KUKA KRL program: EPS_2_25748_MH07A_A_20260121065905.src

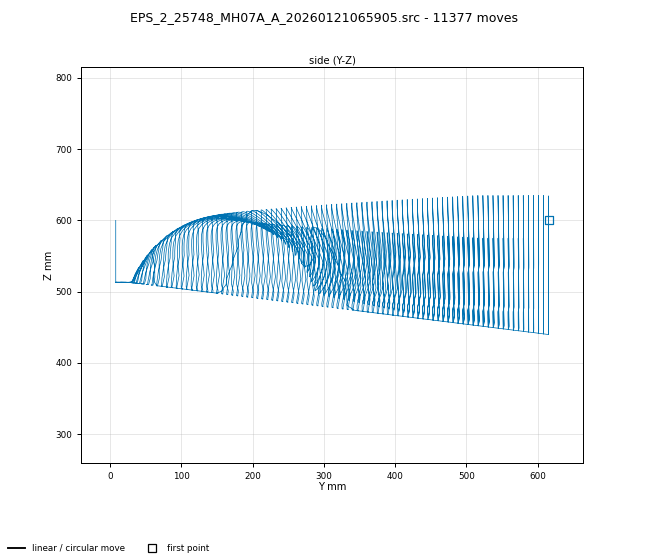
[picture p0: tool path of EPS_2_25748_MH07A_A_20260121065905.src, 11377 of 11379 moves have a stored position in this frame; points joined in program order, loops and branches not executed]
&ACCESS RVP
&REL 4
&COMMENT QRS 19112012
&PARAM EDITMASK = *
DEF PART()
EXT BAS (BAS_COMMAND :IN,REAL :IN )
INT I
BAS (#INITMOV,0 )

;KUKA QRS Post kuka4.cps  Date:22-06-2017 !

File_ID=3007

QRS_PRE_INIT()

;Init var - Until changes are made in qrs_pre_init
Outlet_Square_prg=0
Inlet_1_Square_prg=0
Inlet_2_Square_prg=0
Inlet_3_Square_prg=0
Inlet_4_Square_prg=0
Inlet_5_Square_prg=0

Outlet_1={X 0.000, Y 515.340, Z 534.500, B 0.000, E1 0.000 }
Inlet_1={X 0.000, Y 519.690, Z 474.500, B 0.000, E1 270.000 }
Outlet_1_type=201
Inlet_1_type=201
;QRS#1=Sidecore dimensions
;QRS#2=200-8" PVC SDR 35
;QRS#3=200-8" PVC SDR 35
;QRS#4=
;QRS#5=
;QRS#6=
;QRS#7=
;QRS#8=
;QRS#9=12-08 PSX
;QRS#10=12-08 PSX
;QRS#11=
;QRS#12=
;QRS#13=
;QRS#14=
;QRS#15=
;QRS#16=1220x127x914 3'
;QRS#17=EPS Height
;QRS#18=635
;QRS#19=*
;QRS#20= UPDATED VERSION 22-06-2017
;QRS#21=*
Outlet_Square=0100
Inlet_1_Square=0100
Inlet_2_Square=0
Inlet_3_Square=0
Inlet_4_Square=0
Inlet_5_Square=0
Mill_Square=1
Outlet_Square_Prg=204
Inlet_1_Square_prg=204

QRS_INIT()

$ADVANCE=5

; T1
PTP {E1 173.607,E2 173.607}
PTP {X 0,Y 615.507,A -85,B 0,C 180,E1 173.607,E2 173.607,E3 0,E4 0,E5 0,E6 0}
QRS_SPEED_INIT()
LIN {X 0,Y 615.507,Z 600,A -85,B 0,C 180,E1 173.607,E2 173.607,E3 0,E4 0,E5 0,E6 0} C_VEL
LIN {X 0,Y 615.507,Z 449.87,A -85,B 0,C 180,E1 173.607,E2 173.607} C_VEL
LIN {X 0,Y 615.507,Z 441.69,A -85,B 0,C 180,E1 173.607,E2 173.607} C_VEL
LIN {X 0,Y 615.491,Z 439.69,A -85,B 0,C 180,E1 173.421,E2 173.421} C_VEL
LIN {X 0,Y 615.486,Z 439.701,A -85,B 0,C 180,E1 170.801,E2 170.801} C_VEL
LIN {X 0,Y 615.477,Z 439.696,A -85,B 0,C 180,E1 168.139,E2 168.139} C_VEL
LIN {X 0,Y 615.49,Z 439.69,A -85,B 0,C 180,E1 165.451,E2 165.451} C_VEL
LIN {X 0,Y 615.491,Z 439.693,A -85,B 0,C 180,E1 162.729,E2 162.729} C_VEL
LIN {X 0,Y 615.49,Z 439.702,A -85,B 0,C 180,E1 159.967,E2 159.967} C_VEL
LIN {X 0,Y 615.486,Z 439.695,A -85,B 0,C 180,E1 157.155,E2 157.155} C_VEL
LIN {X 0,Y 615.48,Z 439.693,A -85,B 0,C 180,E1 154.284,E2 154.284} C_VEL
LIN {X 0,Y 615.491,Z 439.69,A -85,B 0,C 180,E1 151.549,E2 151.549} C_VEL
LIN {X 0,Y 615.491,Z 439.699,A -85,B 0,C 180,E1 148.914,E2 148.914} C_VEL
LIN {X 0,Y 615.485,Z 439.692,A -85,B 0,C 180,E1 146.466,E2 146.466} C_VEL
LIN {X 0,Y 615.489,Z 439.69,A -85,B 0,C 180,E1 143.575,E2 143.575} C_VEL
LIN {X 0,Y 615.484,Z 439.696,A -85,B 0,C 180,E1 140.938,E2 140.938} C_VEL
LIN {X 0,Y 615.486,Z 439.693,A -85,B 0,C 180,E1 138.526,E2 138.526} C_VEL
LIN {X 0,Y 615.493,Z 439.689,A -85,B 0,C 180,E1 135.85,E2 135.85} C_VEL
LIN {X 0,Y 615.481,Z 439.695,A -85,B 0,C 180,E1 133.046,E2 133.046} C_VEL
LIN {X 0,Y 615.493,Z 439.695,A -85,B 0,C 180,E1 130.089,E2 130.089} C_VEL
LIN {X 0,Y 615.492,Z 439.7,A -85,B 0,C 180,E1 127.242,E2 127.242} C_VEL
LIN {X 0,Y 615.491,Z 439.69,A -85,B 0,C 180,E1 124.7,E2 124.7} C_VEL
LIN {X 0,Y 615.491,Z 439.697,A -85,B 0,C 180,E1 122.331,E2 122.331} C_VEL
LIN {X 0,Y 615.499,Z 439.691,A -85,B 0,C 180,E1 119.796,E2 119.796} C_VEL
LIN {X 0,Y 615.486,Z 439.69,A -85,B 0,C 180,E1 117.044,E2 117.044} C_VEL
LIN {X 0,Y 615.483,Z 439.693,A -85,B 0,C 180,E1 114.272,E2 114.272} C_VEL
LIN {X 0,Y 615.48,Z 439.7,A -85,B 0,C 180,E1 111.432,E2 111.432} C_VEL
LIN {X 0,Y 615.488,Z 439.699,A -85,B 0,C 180,E1 108.603,E2 108.603} C_VEL
LIN {X 0,Y 615.489,Z 439.691,A -85,B 0,C 180,E1 105.905,E2 105.905} C_VEL
LIN {X 0,Y 615.482,Z 439.692,A -85,B 0,C 180,E1 103.201,E2 103.201} C_VEL
LIN {X 0,Y 615.488,Z 439.698,A -85,B 0,C 180,E1 100.527,E2 100.527} C_VEL
LIN {X 0,Y 615.494,Z 439.693,A -85,B 0,C 180,E1 97.875,E2 97.875} C_VEL
LIN {X 0,Y 615.482,Z 439.691,A -85,B 0,C 180,E1 95.241,E2 95.241} C_VEL
LIN {X 0,Y 615.484,Z 439.697,A -85,B 0,C 180,E1 92.618,E2 92.618} C_VEL
LIN {X 0,Y 615.491,Z 439.695,A -85,B 0,C 180,E1 90,E2 90} C_VEL
LIN {X 0,Y 615.478,Z 439.692,A -85,B 0,C 180,E1 87.382,E2 87.382} C_VEL
LIN {X 0,Y 615.482,Z 439.696,A -85,B 0,C 180,E1 84.759,E2 84.759} C_VEL
LIN {X 0,Y 615.488,Z 439.698,A -85,B 0,C 180,E1 82.124,E2 82.124} C_VEL
LIN {X 0,Y 615.478,Z 439.693,A -85,B 0,C 180,E1 79.473,E2 79.473} C_VEL
LIN {X 0,Y 615.48,Z 439.694,A -85,B 0,C 180,E1 76.798,E2 76.798} C_VEL
LIN {X 0,Y 615.486,Z 439.701,A -85,B 0,C 180,E1 74.095,E2 74.095} C_VEL
LIN {X 0,Y 615.483,Z 439.696,A -85,B 0,C 180,E1 71.354,E2 71.354} C_VEL
LIN {X 0,Y 615.477,Z 439.693,A -85,B 0,C 180,E1 68.568,E2 68.568} C_VEL
LIN {X 0,Y 615.478,Z 439.693,A -85,B 0,C 180,E1 65.727,E2 65.727} C_VEL
LIN {X 0,Y 615.486,Z 439.696,A -85,B 0,C 180,E1 62.956,E2 62.956} C_VEL
LIN {X 0,Y 615.497,Z 439.698,A -85,B 0,C 180,E1 60.205,E2 60.205} C_VEL
LIN {X 0,Y 615.479,Z 439.693,A -85,B 0,C 180,E1 57.542,E2 57.542} C_VEL
LIN {X 0,Y 615.499,Z 439.693,A -85,B 0,C 180,E1 55.185,E2 55.185} C_VEL
LIN {X 0,Y 615.48,Z 439.694,A -85,B 0,C 180,E1 52.757,E2 52.757} C_VEL
LIN {X 0,Y 615.476,Z 439.693,A -85,B 0,C 180,E1 49.913,E2 49.913} C_VEL
LIN {X 0,Y 615.499,Z 439.7,A -85,B 0,C 180,E1 47.648,E2 47.648} C_VEL
LIN {X 0,Y 615.484,Z 439.694,A -85,B 0,C 180,E1 44.931,E2 44.931} C_VEL
LIN {X 0,Y 615.488,Z 439.69,A -85,B 0,C 180,E1 42.08,E2 42.08} C_VEL
LIN {X 0,Y 615.481,Z 439.702,A -85,B 0,C 180,E1 39.751,E2 39.751} C_VEL
LIN {X 0,Y 615.487,Z 439.697,A -85,B 0,C 180,E1 36.936,E2 36.936} C_VEL
LIN {X 0,Y 615.48,Z 439.694,A -85,B 0,C 180,E1 35.617,E2 35.617} C_VEL
LIN {X 0,Y 615.483,Z 440.393,A -85,B 0,C 180,E1 34.7,E2 34.7} C_VEL
LIN {X 0,Y 615.494,Z 443.234,A -85,B 0,C 180,E1 32.331,E2 32.331} C_VEL
LIN {X 0,Y 615.487,Z 446.882,A -85,B 0,C 180,E1 29.407,E2 29.407} C_VEL
LIN {X 0,Y 615.481,Z 449.92,A -85,B 0,C 180,E1 27.043,E2 27.043} C_VEL
LIN {X 0,Y 615.493,Z 453.568,A -85,B 0,C 180,E1 24.272,E2 24.272} C_VEL
LIN {X 0,Y 615.494,Z 457.377,A -85,B 0,C 180,E1 21.432,E2 21.432} C_VEL
LIN {X 0,Y 615.494,Z 461.252,A -85,B 0,C 180,E1 18.605,E2 18.605} C_VEL
LIN {X 0,Y 615.476,Z 465.011,A -85,B 0,C 180,E1 15.906,E2 15.906} C_VEL
LIN {X 0,Y 615.493,Z 468.827,A -85,B 0,C 180,E1 13.201,E2 13.201} C_VEL
LIN {X 0,Y 615.484,Z 471.187,A -85,B 0,C 180,E1 11.548,E2 11.548} C_VEL
LIN {X 0,Y 615.485,Z 486.249,A -85,B 0,C 180,E1 11.193,E2 11.193} C_VEL
LIN {X 0,Y 615.481,Z 498.967,A -85,B 0,C 180,E1 10.749,E2 10.749} C_VEL
LIN {X 0,Y 615.483,Z 510.755,A -85,B 0,C 180,E1 10.195,E2 10.195} C_VEL
LIN {X 0,Y 615.498,Z 521.845,A -85,B 0,C 180,E1 9.53,E2 9.53} C_VEL
LIN {X 0,Y 615.498,Z 530.82,A -85,B 0,C 180,E1 8.868,E2 8.868} C_VEL
LIN {X 0,Y 615.498,Z 540.032,A -85,B 0,C 180,E1 8.041,E2 8.041} C_VEL
LIN {X 0,Y 615.499,Z 548.89,A -85,B 0,C 180,E1 7.058,E2 7.058} C_VEL
LIN {X 0,Y 615.497,Z 556.122,A -85,B 0,C 180,E1 6.063,E2 6.063} C_VEL
LIN {X 0,Y 615.497,Z 560.957,A -85,B 0,C 180,E1 5.241,E2 5.241} C_VEL
LIN {X 0,Y 615.493,Z 565.657,A -85,B 0,C 180,E1 4.257,E2 4.257} C_VEL
LIN {X 0,Y 615.495,Z 569.254,A -85,B 0,C 180,E1 3.273,E2 3.273} C_VEL
LIN {X 0,Y 615.496,Z 571.114,A -85,B 0,C 180,E1 2.618,E2 2.618} C_VEL
LIN {X 0,Y 615.497,Z 572.533,A -85,B 0,C 180,E1 1.963,E2 1.963} C_VEL
LIN {X 0,Y 615.497,Z 574.141,A -85,B 0,C 180,E1 0.654,E2 0.654} C_VEL
LIN {X 0,Y 615.494,Z 574.384,A -85,B 0,C 180,E1 0,E2 0} C_VEL
LIN {X 0,Y 615.495,Z 574.206,A -85,B 0,C 180,E1 -0.654,E2 -0.654} C_VEL
LIN {X 0,Y 615.496,Z 572.683,A -85,B 0,C 180,E1 -1.963,E2 -1.963} C_VEL
LIN {X 0,Y 615.498,Z 571.341,A -85,B 0,C 180,E1 -2.618,E2 -2.618} C_VEL
LIN {X 0,Y 615.498,Z 568.494,A -85,B 0,C 180,E1 -3.601,E2 -3.601} C_VEL
LIN {X 0,Y 615.498,Z 564.635,A -85,B 0,C 180,E1 -4.584,E2 -4.584} C_VEL
LIN {X 0,Y 615.499,Z 559.652,A -85,B 0,C 180,E1 -5.57,E2 -5.57} C_VEL
LIN {X 0,Y 615.496,Z 553.208,A -85,B 0,C 180,E1 -6.582,E2 -6.582} C_VEL
LIN {X 0,Y 615.497,Z 545.537,A -85,B 0,C 180,E1 -7.545,E2 -7.545} C_VEL
LIN {X 0,Y 615.498,Z 535.759,A -85,B 0,C 180,E1 -8.536,E2 -8.536} C_VEL
LIN {X 0,Y 615.498,Z 525.494,A -85,B 0,C 180,E1 -9.364,E2 -9.364} C_VEL
LIN {X 0,Y 615.479,Z 513.933,A -85,B 0,C 180,E1 -10.111,E2 -10.111} C_VEL
LIN {X 0,Y 615.482,Z 502.146,A -85,B 0,C 180,E1 -10.704,E2 -10.704} C_VEL
LIN {X 0,Y 615.483,Z 489.162,A -85,B 0,C 180,E1 -11.193,E2 -11.193} C_VEL
LIN {X 0,Y 615.487,Z 476.561,A -85,B 0,C 180,E1 -11.527,E2 -11.527} C_VEL
LIN {X 0,Y 615.484,Z 471.197,A -85,B 0,C 180,E1 -11.631,E2 -11.631} C_VEL
LIN {X 0,Y 615.476,Z 467.929,A -85,B 0,C 180,E1 -13.927,E2 -13.927} C_VEL
LIN {X 0,Y 615.487,Z 464.181,A -85,B 0,C 180,E1 -16.587,E2 -16.587} C_VEL
LIN {X 0,Y 615.489,Z 460.369,A -85,B 0,C 180,E1 -19.338,E2 -19.338} C_VEL
LIN {X 0,Y 615.479,Z 456.548,A -85,B 0,C 180,E1 -22.137,E2 -22.137} C_VEL
LIN {X 0,Y 615.491,Z 453.686,A -85,B 0,C 180,E1 -24.272,E2 -24.272} C_VEL
LIN {X 0,Y 615.481,Z 449.862,A -85,B 0,C 180,E1 -27.178,E2 -27.178} C_VEL
LIN {X 0,Y 615.497,Z 446.505,A -85,B 0,C 180,E1 -29.796,E2 -29.796} C_VEL
LIN {X 0,Y 615.489,Z 443.245,A -85,B 0,C 180,E1 -32.457,E2 -32.457} C_VEL
LIN {X 0,Y 615.488,Z 440.551,A -85,B 0,C 180,E1 -34.815,E2 -34.815} C_VEL
LIN {X 0,Y 615.478,Z 439.698,A -85,B 0,C 180,E1 -35.832,E2 -35.832} C_VEL
LIN {X 0,Y 615.491,Z 439.697,A -85,B 0,C 180,E1 -38.068,E2 -38.068} C_VEL
LIN {X 0,Y 615.479,Z 439.698,A -85,B 0,C 180,E1 -40.607,E2 -40.607} C_VEL
LIN {X 0,Y 615.498,Z 439.693,A -85,B 0,C 180,E1 -43.244,E2 -43.244} C_VEL
LIN {X 0,Y 615.483,Z 439.698,A -85,B 0,C 180,E1 -46.003,E2 -46.003} C_VEL
LIN {X 0,Y 615.493,Z 439.697,A -85,B 0,C 180,E1 -48.905,E2 -48.905} C_VEL
LIN {X 0,Y 615.492,Z 439.701,A -85,B 0,C 180,E1 -51.096,E2 -51.096} C_VEL
LIN {X 0,Y 615.484,Z 439.703,A -85,B 0,C 180,E1 -53.575,E2 -53.575} C_VEL
LIN {X 0,Y 615.486,Z 439.895,A -85,B 0,C 180,E1 -54.484,E2 -54.484} C_VEL
LIN {X 0,Y 615.486,Z 448.578,A -85,B 0,C 180,E1 -57.154,E2 -57.154} C_VEL
LIN {X 0,Y 615.48,Z 457.828,A -85,B 0,C 180,E1 -59.839,E2 -59.839} C_VEL
LIN {X 0,Y 615.481,Z 467.078,A -85,B 0,C 180,E1 -62.454,E2 -62.454} C_VEL
LIN {X 0,Y 615.488,Z 476.316,A -85,B 0,C 180,E1 -65.008,E2 -65.008} C_VEL
LIN {X 0,Y 615.482,Z 486.871,A -85,B 0,C 180,E1 -67.863,E2 -67.863} C_VEL
LIN {X 0,Y 615.475,Z 497.419,A -85,B 0,C 180,E1 -70.662,E2 -70.662} C_VEL
LIN {X 0,Y 615.48,Z 507.958,A -85,B 0,C 180,E1 -73.413,E2 -73.413} C_VEL
LIN {X 0,Y 615.493,Z 518.494,A -85,B 0,C 180,E1 -76.126,E2 -76.126} C_VEL
LIN {X 0,Y 615.487,Z 527.208,A -85,B 0,C 180,E1 -78.348,E2 -78.348} C_VEL
LIN {X 0,Y 615.496,Z 541.817,A -85,B 0,C 180,E1 -78.64,E2 -78.64} C_VEL
LIN {X 0,Y 615.49,Z 554.557,A -85,B 0,C 180,E1 -79.036,E2 -79.036} C_VEL
LIN {X 0,Y 615.477,Z 566.765,A -85,B 0,C 180,E1 -79.556,E2 -79.556} C_VEL
LIN {X 0,Y 615.491,Z 577.386,A -85,B 0,C 180,E1 -80.138,E2 -80.138} C_VEL
LIN {X 0,Y 615.498,Z 588.23,A -85,B 0,C 180,E1 -80.884,E2 -80.884} C_VEL
LIN {X 0,Y 615.497,Z 598.81,A -85,B 0,C 180,E1 -81.794,E2 -81.794} C_VEL
LIN {X 0,Y 615.498,Z 606.605,A -85,B 0,C 180,E1 -82.619,E2 -82.619} C_VEL
LIN {X 0,Y 615.496,Z 614.202,A -85,B 0,C 180,E1 -83.608,E2 -83.608} C_VEL
LIN {X 0,Y 615.498,Z 621.204,A -85,B 0,C 180,E1 -84.759,E2 -84.759} C_VEL
LIN {X 0,Y 615.493,Z 625.851,A -85,B 0,C 180,E1 -85.743,E2 -85.743} C_VEL
LIN {X 0,Y 615.495,Z 629.398,A -85,B 0,C 180,E1 -86.727,E2 -86.727} C_VEL
LIN {X 0,Y 615.497,Z 631.233,A -85,B 0,C 180,E1 -87.382,E2 -87.382} C_VEL
LIN {X 0,Y 615.497,Z 632.608,A -85,B 0,C 180,E1 -88.037,E2 -88.037} C_VEL
LIN {X 0,Y 615.496,Z 634.173,A -85,B 0,C 180,E1 -89.346,E2 -89.346} C_VEL
LIN {X 0,Y 615.494,Z 634.389,A -85,B 0,C 180,E1 -90,E2 -90} C_VEL
LIN {X 0,Y 615.496,Z 633.58,A -85,B 0,C 180,E1 -91.309,E2 -91.309} C_VEL
LIN {X 0,Y 615.497,Z 632.608,A -85,B 0,C 180,E1 -91.963,E2 -91.963} C_VEL
LIN {X 0,Y 615.497,Z 631.233,A -85,B 0,C 180,E1 -92.618,E2 -92.618} C_VEL
LIN {X 0,Y 615.496,Z 628.35,A -85,B 0,C 180,E1 -93.601,E2 -93.601} C_VEL
LIN {X 0,Y 615.498,Z 624.442,A -85,B 0,C 180,E1 -94.584,E2 -94.584} C_VEL
LIN {X 0,Y 615.499,Z 619.405,A -85,B 0,C 180,E1 -95.57,E2 -95.57} C_VEL
LIN {X 0,Y 615.497,Z 612.869,A -85,B 0,C 180,E1 -96.583,E2 -96.583} C_VEL
LIN {X 0,Y 615.497,Z 605.133,A -85,B 0,C 180,E1 -97.545,E2 -97.545} C_VEL
LIN {X 0,Y 615.498,Z 597.045,A -85,B 0,C 180,E1 -98.371,E2 -98.371} C_VEL
LIN {X 0,Y 615.499,Z 587.168,A -85,B 0,C 180,E1 -99.199,E2 -99.199} C_VEL
LIN {X 0,Y 615.488,Z 575.982,A -85,B 0,C 180,E1 -99.945,E2 -99.945} C_VEL
LIN {X 0,Y 615.478,Z 565.025,A -85,B 0,C 180,E1 -100.527,E2 -100.527} C_VEL
LIN {X 0,Y 615.494,Z 552.486,A -85,B 0,C 180,E1 -101.04,E2 -101.04} C_VEL
LIN {X 0,Y 615.495,Z 540.065,A -85,B 0,C 180,E1 -101.401,E2 -101.401} C_VEL
LIN {X 0,Y 615.487,Z 527.209,A -85,B 0,C 180,E1 -101.652,E2 -101.652} C_VEL
LIN {X 0,Y 615.48,Z 517.063,A -85,B 0,C 180,E1 -104.242,E2 -104.242} C_VEL
LIN {X 0,Y 615.495,Z 506.638,A -85,B 0,C 180,E1 -106.928,E2 -106.928} C_VEL
LIN {X 0,Y 615.485,Z 496.105,A -85,B 0,C 180,E1 -109.685,E2 -109.685} C_VEL
LIN {X 0,Y 615.477,Z 486.101,A -85,B 0,C 180,E1 -112.343,E2 -112.343} C_VEL
LIN {X 0,Y 615.489,Z 476.316,A -85,B 0,C 180,E1 -114.992,E2 -114.992} C_VEL
LIN {X 0,Y 615.481,Z 467.079,A -85,B 0,C 180,E1 -117.546,E2 -117.546} C_VEL
LIN {X 0,Y 615.483,Z 457.829,A -85,B 0,C 180,E1 -120.16,E2 -120.16} C_VEL
LIN {X 0,Y 615.489,Z 448.579,A -85,B 0,C 180,E1 -122.846,E2 -122.846} C_VEL
LIN {X 0,Y 615.486,Z 439.694,A -85,B 0,C 180,E1 -125.541,E2 -125.541} C_VEL
LIN {X 0,Y 615.485,Z 439.697,A -85,B 0,C 180,E1 -128.069,E2 -128.069} C_VEL
LIN {X 0,Y 615.484,Z 439.691,A -85,B 0,C 180,E1 -130.607,E2 -130.607} C_VEL
LIN {X 0,Y 615.477,Z 439.698,A -85,B 0,C 180,E1 -133.246,E2 -133.246} C_VEL
LIN {X 0,Y 615.49,Z 439.7,A -85,B 0,C 180,E1 -136.002,E2 -136.002} C_VEL
LIN {X 0,Y 615.485,Z 439.691,A -85,B 0,C 180,E1 -138.526,E2 -138.526} C_VEL
LIN {X 0,Y 615.478,Z 439.697,A -85,B 0,C 180,E1 -141.095,E2 -141.095} C_VEL
LIN {X 0,Y 615.488,Z 439.695,A -85,B 0,C 180,E1 -143.575,E2 -143.575} C_VEL
LIN {X 0,Y 615.484,Z 439.692,A -85,B 0,C 180,E1 -146.466,E2 -146.466} C_VEL
LIN {X 0,Y 615.478,Z 439.694,A -85,B 0,C 180,E1 -149.08,E2 -149.08} C_VEL
LIN {X 0,Y 615.491,Z 439.698,A -85,B 0,C 180,E1 -151.549,E2 -151.549} C_VEL
LIN {X 0,Y 615.485,Z 439.694,A -85,B 0,C 180,E1 -154.432,E2 -154.432} C_VEL
LIN {X 0,Y 615.475,Z 439.693,A -85,B 0,C 180,E1 -157.155,E2 -157.155} C_VEL
LIN {X 0,Y 615.491,Z 439.701,A -85,B 0,C 180,E1 -159.443,E2 -159.443} C_VEL
LIN {X 0,Y 615.477,Z 439.693,A -85,B 0,C 180,E1 -162.043,E2 -162.043} C_VEL
LIN {X 0,Y 615.486,Z 439.691,A -85,B 0,C 180,E1 -164.774,E2 -164.774} C_VEL
LIN {X 0,Y 615.489,Z 439.697,A -85,B 0,C 180,E1 -167.47,E2 -167.47} C_VEL
LIN {X 0,Y 615.479,Z 439.697,A -85,B 0,C 180,E1 -170.138,E2 -170.138} C_VEL
LIN {X 0,Y 615.483,Z 439.691,A -85,B 0,C 180,E1 -172.784,E2 -172.784} C_VEL
LIN {X 0,Y 615.491,Z 439.694,A -85,B 0,C 180,E1 -175.416,E2 -175.416} C_VEL
LIN {X 0,Y 615.482,Z 439.699,A -85,B 0,C 180,E1 -178.037,E2 -178.037} C_VEL
LIN {X 0,Y 615.488,Z 439.69,A -85,B 0,C 180,E1 -180.654,E2 -180.654} C_VEL
LIN {X 0,Y 615.485,Z 439.694,A -85,B 0,C 180,E1 -183.273,E2 -183.273} C_VEL
LIN {X 0,Y 615.485,Z 439.7,A -85,B 0,C 180,E1 -185.899,E2 -185.899} C_VEL
LIN {X 0,Y 615.491,Z 439.69,A -85,B 0,C 180,E1 -186.579,E2 -186.579} C_VEL
LIN {X 0,Y 614.811,Z 439.842,A -85,B 0,C 180,E1 -187.125,E2 -187.125} C_VEL
LIN {X 0,Y 611.975,Z 440.254,A -85,B 0,C 180,E1 -188.011,E2 -188.011} C_VEL
LIN {X 0,Y 609.584,Z 440.567,A -85,B 0,C 180,E1 -188.724,E2 -188.724} C_VEL
LIN {X 0,Y 608.548,Z 440.685,A -85,B 0,C 180,E1 -189.273,E2 -189.273} C_VEL
LIN {X 0,Y 608.457,Z 440.693,A -85,B 0,C 180,E1 -189.459,E2 -189.459} C_VEL
LIN {X 0,Y 608.457,Z 440.694,A -85,B 0,C 180,E1 -192,E2 -192} C_VEL
LIN {X 0,Y 608.478,Z 440.689,A -85,B 0,C 180,E1 -194.721,E2 -194.721} C_VEL
LIN {X 0,Y 608.453,Z 440.692,A -85,B 0,C 180,E1 -197.477,E2 -197.477} C_VEL
LIN {X 0,Y 608.465,Z 440.693,A -85,B 0,C 180,E1 -200.274,E2 -200.274} C_VEL
LIN {X 0,Y 608.462,Z 440.69,A -85,B 0,C 180,E1 -202.477,E2 -202.477} C_VEL
LIN {X 0,Y 608.448,Z 440.693,A -85,B 0,C 180,E1 -205.301,E2 -205.301} C_VEL
LIN {X 0,Y 608.449,Z 440.694,A -85,B 0,C 180,E1 -207.518,E2 -207.518} C_VEL
LIN {X 0,Y 608.464,Z 440.691,A -85,B 0,C 180,E1 -209.971,E2 -209.971} C_VEL
LIN {X 0,Y 608.463,Z 440.692,A -85,B 0,C 180,E1 -212.88,E2 -212.88} C_VEL
LIN {X 0,Y 608.446,Z 440.694,A -85,B 0,C 180,E1 -215.278,E2 -215.278} C_VEL
LIN {X 0,Y 608.469,Z 440.69,A -85,B 0,C 180,E1 -217.747,E2 -217.747} C_VEL
LIN {X 0,Y 608.448,Z 440.699,A -85,B 0,C 180,E1 -220.328,E2 -220.328} C_VEL
LIN {X 0,Y 608.452,Z 440.693,A -85,B 0,C 180,E1 -222.96,E2 -222.96} C_VEL
LIN {X 0,Y 608.45,Z 440.692,A -85,B 0,C 180,E1 -225.737,E2 -225.737} C_VEL
LIN {X 0,Y 608.457,Z 440.692,A -85,B 0,C 180,E1 -228.659,E2 -228.659} C_VEL
LIN {X 0,Y 608.466,Z 440.691,A -85,B 0,C 180,E1 -231.761,E2 -231.761} C_VEL
LIN {X 0,Y 608.451,Z 440.693,A -85,B 0,C 180,E1 -233.955,E2 -233.955} C_VEL
LIN {X 0,Y 608.453,Z 440.693,A -85,B 0,C 180,E1 -236.329,E2 -236.329} C_VEL
LIN {X 0,Y 608.451,Z 440.694,A -85,B 0,C 180,E1 -238.733,E2 -238.733} C_VEL
LIN {X 0,Y 608.47,Z 440.689,A -85,B 0,C 180,E1 -241.382,E2 -241.382} C_VEL
LIN {X 0,Y 608.446,Z 440.696,A -85,B 0,C 180,E1 -243.965,E2 -243.965} C_VEL
LIN {X 0,Y 608.467,Z 440.69,A -85,B 0,C 180,E1 -246.155,E2 -246.155} C_VEL
LIN {X 0,Y 608.457,Z 440.691,A -85,B 0,C 180,E1 -249.019,E2 -249.019} C_VEL
LIN {X 0,Y 608.457,Z 440.694,A -85,B 0,C 180,E1 -251.828,E2 -251.828} C_VEL
LIN {X 0,Y 608.473,Z 440.695,A -85,B 0,C 180,E1 -254.594,E2 -254.594} C_VEL
LIN {X 0,Y 608.472,Z 440.69,A -85,B 0,C 180,E1 -257.323,E2 -257.323} C_VEL
LIN {X 0,Y 608.462,Z 440.69,A -85,B 0,C 180,E1 -260.023,E2 -260.023} C_VEL
LIN {X 0,Y 608.466,Z 440.693,A -85,B 0,C 180,E1 -262.701,E2 -262.701} C_VEL
LIN {X 0,Y 608.452,Z 440.695,A -85,B 0,C 180,E1 -265.362,E2 -265.362} C_VEL
LIN {X 0,Y 608.468,Z 440.69,A -85,B 0,C 180,E1 -268.014,E2 -268.014} C_VEL
LIN {X 0,Y 608.475,Z 440.69,A -85,B 0,C 180,E1 -270.662,E2 -270.662} C_VEL
LIN {X 0,Y 608.48,Z 440.694,A -85,B 0,C 180,E1 -273.311,E2 -273.311} C_VEL
LIN {X 0,Y 608.467,Z 440.69,A -85,B 0,C 180,E1 -275.967,E2 -275.967} C_VEL
LIN {X 0,Y 608.452,Z 440.692,A -85,B 0,C 180,E1 -278.636,E2 -278.636} C_VEL
LIN {X 0,Y 608.486,Z 440.692,A -85,B 0,C 180,E1 -281.324,E2 -281.324} C_VEL
LIN {X 0,Y 608.476,Z 440.692,A -85,B 0,C 180,E1 -284.037,E2 -284.037} C_VEL
LIN {X 0,Y 608.444,Z 440.693,A -85,B 0,C 180,E1 -286.784,E2 -286.784} C_VEL
LIN {X 0,Y 608.45,Z 440.692,A -85,B 0,C 180,E1 -289.571,E2 -289.571} C_VEL
LIN {X 0,Y 608.465,Z 440.692,A -85,B 0,C 180,E1 -292.406,E2 -292.406} C_VEL
LIN {X 0,Y 608.453,Z 440.692,A -85,B 0,C 180,E1 -294.571,E2 -294.571} C_VEL
LIN {X 0,Y 608.477,Z 440.69,A -85,B 0,C 180,E1 -297.206,E2 -297.206} C_VEL
LIN {X 0,Y 608.472,Z 440.695,A -85,B 0,C 180,E1 -299.971,E2 -299.971} C_VEL
LIN {X 0,Y 608.455,Z 440.696,A -85,B 0,C 180,E1 -302.88,E2 -302.88} C_VEL
LIN {X 0,Y 608.447,Z 440.692,A -85,B 0,C 180,E1 -305.278,E2 -305.278} C_VEL
LIN {X 0,Y 608.467,Z 440.695,A -85,B 0,C 180,E1 -307.747,E2 -307.747} C_VEL
LIN {X 0,Y 608.444,Z 440.694,A -85,B 0,C 180,E1 -310.328,E2 -310.328} C_VEL
LIN {X 0,Y 608.45,Z 440.692,A -85,B 0,C 180,E1 -312.96,E2 -312.96} C_VEL
LIN {X 0,Y 608.46,Z 440.694,A -85,B 0,C 180,E1 -315.736,E2 -315.736} C_VEL
LIN {X 0,Y 608.465,Z 440.696,A -85,B 0,C 180,E1 -318.658,E2 -318.658} C_VEL
LIN {X 0,Y 608.466,Z 440.696,A -85,B 0,C 180,E1 -321.76,E2 -321.76} C_VEL
LIN {X 0,Y 608.449,Z 440.692,A -85,B 0,C 180,E1 -323.955,E2 -323.955} C_VEL
LIN {X 0,Y 608.423,Z 440.996,A -85,B 0,C 180,E1 -325.099,E2 -325.099} C_VEL
LIN {X 0,Y 608.435,Z 443.838,A -85,B 0,C 180,E1 -327.482,E2 -327.482} C_VEL
LIN {X 0,Y 608.444,Z 447.196,A -85,B 0,C 180,E1 -330.219,E2 -330.219} C_VEL
LIN {X 0,Y 608.427,Z 450.493,A -85,B 0,C 180,E1 -332.803,E2 -332.803} C_VEL
LIN {X 0,Y 608.423,Z 453.921,A -85,B 0,C 180,E1 -335.427,E2 -335.427} C_VEL
LIN {X 0,Y 608.418,Z 457.764,A -85,B 0,C 180,E1 -338.306,E2 -338.306} C_VEL
LIN {X 0,Y 608.424,Z 461.607,A -85,B 0,C 180,E1 -341.129,E2 -341.129} C_VEL
LIN {X 0,Y 608.421,Z 465.45,A -85,B 0,C 180,E1 -343.905,E2 -343.905} C_VEL
LIN {X 0,Y 608.432,Z 469.294,A -85,B 0,C 180,E1 -346.643,E2 -346.643} C_VEL
LIN {X 0,Y 608.429,Z 471.666,A -85,B 0,C 180,E1 -348.316,E2 -348.316} C_VEL
LIN {X 0,Y 608.53,Z 487.61,A -85,B 0,C 180,E1 -348.714,E2 -348.714} C_VEL
LIN {X 0,Y 608.503,Z 500.162,A -85,B 0,C 180,E1 -349.171,E2 -349.171} C_VEL
LIN {X 0,Y 608.48,Z 512.497,A -85,B 0,C 180,E1 -349.771,E2 -349.771} C_VEL
LIN {X 0,Y 608.488,Z 523.302,A -85,B 0,C 180,E1 -350.443,E2 -350.443} C_VEL
LIN {X 0,Y 608.477,Z 533.075,A -85,B 0,C 180,E1 -351.197,E2 -351.197} C_VEL
LIN {X 0,Y 608.46,Z 541.974,A -85,B 0,C 180,E1 -352.033,E2 -352.033} C_VEL
LIN {X 0,Y 608.465,Z 550.661,A -85,B 0,C 180,E1 -353.034,E2 -353.034} C_VEL
LIN {X 0,Y 608.439,Z 557.592,A -85,B 0,C 180,E1 -354.033,E2 -354.033} C_VEL
LIN {X 0,Y 608.436,Z 563.146,A -85,B 0,C 180,E1 -355.03,E2 -355.03} C_VEL
LIN {X 0,Y 608.434,Z 567.508,A -85,B 0,C 180,E1 -356.026,E2 -356.026} C_VEL
LIN {X 0,Y 608.426,Z 569.812,A -85,B 0,C 180,E1 -356.689,E2 -356.689} C_VEL
LIN {X 0,Y 608.425,Z 571.69,A -85,B 0,C 180,E1 -357.352,E2 -357.352} C_VEL
LIN {X 0,Y 608.442,Z 573.126,A -85,B 0,C 180,E1 -358.014,E2 -358.014} C_VEL
LIN {X 0,Y 608.44,Z 574.752,A -85,B 0,C 180,E1 -359.338,E2 -359.338} C_VEL
LIN {X 0,Y 608.434,Z 574.995,A -85,B 0,C 180,E1 -360,E2 -360} C_VEL
LIN {X 0,Y 608.438,Z 574.815,A -85,B 0,C 180,E1 -360.662,E2 -360.662} C_VEL
LIN {X 0,Y 608.441,Z 573.276,A -85,B 0,C 180,E1 -361.986,E2 -361.986} C_VEL
LIN {X 0,Y 608.426,Z 571.919,A -85,B 0,C 180,E1 -362.648,E2 -362.648} C_VEL
LIN {X 0,Y 608.45,Z 569.042,A -85,B 0,C 180,E1 -363.642,E2 -363.642} C_VEL
LIN {X 0,Y 608.433,Z 565.143,A -85,B 0,C 180,E1 -364.638,E2 -364.638} C_VEL
LIN {X 0,Y 608.45,Z 560.112,A -85,B 0,C 180,E1 -365.634,E2 -365.634} C_VEL
LIN {X 0,Y 608.441,Z 553.795,A -85,B 0,C 180,E1 -366.633,E2 -366.633} C_VEL
LIN {X 0,Y 608.475,Z 545.879,A -85,B 0,C 180,E1 -367.633,E2 -367.633} C_VEL
LIN {X 0,Y 608.472,Z 536.037,A -85,B 0,C 180,E1 -368.636,E2 -368.636} C_VEL
LIN {X 0,Y 608.48,Z 525.715,A -85,B 0,C 180,E1 -369.473,E2 -369.473} C_VEL
LIN {X 0,Y 608.477,Z 514.1,A -85,B 0,C 180,E1 -370.229,E2 -370.229} C_VEL
LIN {X 0,Y 608.502,Z 502.088,A -85,B 0,C 180,E1 -370.836,E2 -370.836} C_VEL
LIN {X 0,Y 608.529,Z 489.263,A -85,B 0,C 180,E1 -371.323,E2 -371.323} C_VEL
LIN {X 0,Y 608.535,Z 476.647,A -85,B 0,C 180,E1 -371.66,E2 -371.66} C_VEL
LIN {X 0,Y 608.429,Z 471.674,A -85,B 0,C 180,E1 -371.768,E2 -371.768} C_VEL
LIN {X 0,Y 608.42,Z 468.46,A -85,B 0,C 180,E1 -374.039,E2 -374.039} C_VEL
LIN {X 0,Y 608.419,Z 464.615,A -85,B 0,C 180,E1 -376.785,E2 -376.785} C_VEL
LIN {X 0,Y 608.412,Z 460.77,A -85,B 0,C 180,E1 -379.572,E2 -379.572} C_VEL
LIN {X 0,Y 608.432,Z 456.84,A -85,B 0,C 180,E1 -382.469,E2 -382.469} C_VEL
LIN {X 0,Y 608.427,Z 453.078,A -85,B 0,C 180,E1 -385.302,E2 -385.302} C_VEL
LIN {X 0,Y 608.435,Z 449.233,A -85,B 0,C 180,E1 -388.268,E2 -388.268} C_VEL
LIN {X 0,Y 608.43,Z 446.348,A -85,B 0,C 180,E1 -390.547,E2 -390.547} C_VEL
LIN {X 0,Y 608.435,Z 443.668,A -85,B 0,C 180,E1 -392.881,E2 -392.881} C_VEL
LIN {X 0,Y 608.442,Z 440.88,A -85,B 0,C 180,E1 -395.278,E2 -395.278} C_VEL
LIN {X 0,Y 608.474,Z 440.695,A -85,B 0,C 180,E1 -397.746,E2 -397.746} C_VEL
LIN {X 0,Y 608.45,Z 440.698,A -85,B 0,C 180,E1 -400.328,E2 -400.328} C_VEL
LIN {X 0,Y 608.485,Z 440.69,A -85,B 0,C 180,E1 -403.31,E2 -403.31} C_VEL
LIN {X 0,Y 608.468,Z 440.695,A -85,B 0,C 180,E1 -406.13,E2 -406.13} C_VEL
LIN {X 0,Y 608.461,Z 440.696,A -85,B 0,C 180,E1 -408.824,E2 -408.824} C_VEL
LIN {X 0,Y 608.472,Z 440.693,A -85,B 0,C 180,E1 -411.412,E2 -411.412} C_VEL
LIN {X 0,Y 608.48,Z 440.695,A -85,B 0,C 180,E1 -414.228,E2 -414.228} C_VEL
LIN {X 0,Y 608.523,Z 447.254,A -85,B 0,C 180,E1 -416.333,E2 -416.333} C_VEL
LIN {X 0,Y 608.521,Z 456.595,A -85,B 0,C 180,E1 -419.09,E2 -419.09} C_VEL
LIN {X 0,Y 608.483,Z 465.803,A -85,B 0,C 180,E1 -421.735,E2 -421.735} C_VEL
LIN {X 0,Y 608.492,Z 474.859,A -85,B 0,C 180,E1 -424.276,E2 -424.276} C_VEL
LIN {X 0,Y 608.462,Z 484.337,A -85,B 0,C 180,E1 -426.876,E2 -426.876} C_VEL
LIN {X 0,Y 608.465,Z 493.418,A -85,B 0,C 180,E1 -429.323,E2 -429.323} C_VEL
LIN {X 0,Y 608.449,Z 504.196,A -85,B 0,C 180,E1 -432.176,E2 -432.176} C_VEL
LIN {X 0,Y 608.442,Z 514.787,A -85,B 0,C 180,E1 -434.936,E2 -434.936} C_VEL
LIN {X 0,Y 608.443,Z 525.378,A -85,B 0,C 180,E1 -437.661,E2 -437.661} C_VEL
LIN {X 0,Y 608.443,Z 527.53,A -85,B 0,C 180,E1 -438.211,E2 -438.211} C_VEL
LIN {X 0,Y 608.542,Z 542.692,A -85,B 0,C 180,E1 -438.53,E2 -438.53} C_VEL
LIN {X 0,Y 608.526,Z 554.276,A -85,B 0,C 180,E1 -438.894,E2 -438.894} C_VEL
LIN {X 0,Y 608.506,Z 566.919,A -85,B 0,C 180,E1 -439.435,E2 -439.435} C_VEL
LIN {X 0,Y 608.483,Z 577.577,A -85,B 0,C 180,E1 -440.023,E2 -440.023} C_VEL
LIN {X 0,Y 608.483,Z 588.473,A -85,B 0,C 180,E1 -440.778,E2 -440.778} C_VEL
LIN {X 0,Y 608.475,Z 599.111,A -85,B 0,C 180,E1 -441.699,E2 -441.699} C_VEL
LIN {X 0,Y 608.471,Z 606.959,A -85,B 0,C 180,E1 -442.534,E2 -442.534} C_VEL
LIN {X 0,Y 608.461,Z 614.286,A -85,B 0,C 180,E1 -443.484,E2 -443.484} C_VEL
LIN {X 0,Y 608.45,Z 619.865,A -85,B 0,C 180,E1 -444.365,E2 -444.365} C_VEL
LIN {X 0,Y 608.432,Z 624.95,A -85,B 0,C 180,E1 -445.362,E2 -445.362} C_VEL
LIN {X 0,Y 608.449,Z 628.896,A -85,B 0,C 180,E1 -446.358,E2 -446.358} C_VEL
LIN {X 0,Y 608.425,Z 631.809,A -85,B 0,C 180,E1 -447.352,E2 -447.352} C_VEL
LIN {X 0,Y 608.443,Z 633.201,A -85,B 0,C 180,E1 -448.014,E2 -448.014} C_VEL
LIN {X 0,Y 608.438,Z 634.783,A -85,B 0,C 180,E1 -449.338,E2 -449.338} C_VEL
LIN {X 0,Y 608.434,Z 635,A -85,B 0,C 180,E1 -450,E2 -450} C_VEL
LIN {X 0,Y 608.448,Z 634.184,A -85,B 0,C 180,E1 -451.324,E2 -451.324} C_VEL
LIN {X 0,Y 608.442,Z 633.201,A -85,B 0,C 180,E1 -451.986,E2 -451.986} C_VEL
LIN {X 0,Y 608.425,Z 631.809,A -85,B 0,C 180,E1 -452.648,E2 -452.648} C_VEL
LIN {X 0,Y 608.449,Z 628.896,A -85,B 0,C 180,E1 -453.642,E2 -453.642} C_VEL
LIN {X 0,Y 608.432,Z 624.95,A -85,B 0,C 180,E1 -454.638,E2 -454.638} C_VEL
LIN {X 0,Y 608.437,Z 618.877,A -85,B 0,C 180,E1 -455.801,E2 -455.801} C_VEL
LIN {X 0,Y 608.462,Z 612.235,A -85,B 0,C 180,E1 -456.799,E2 -456.799} C_VEL
LIN {X 0,Y 608.455,Z 603.989,A -85,B 0,C 180,E1 -457.8,E2 -457.8} C_VEL
LIN {X 0,Y 608.472,Z 595.537,A -85,B 0,C 180,E1 -458.636,E2 -458.636} C_VEL
LIN {X 0,Y 608.48,Z 585.091,A -85,B 0,C 180,E1 -459.473,E2 -459.473} C_VEL
LIN {X 0,Y 608.494,Z 574.756,A -85,B 0,C 180,E1 -460.145,E2 -460.145} C_VEL
LIN {X 0,Y 608.51,Z 563.266,A -85,B 0,C 180,E1 -460.74,E2 -460.74} C_VEL
LIN {X 0,Y 608.537,Z 550.911,A -85,B 0,C 180,E1 -461.224,E2 -461.224} C_VEL
LIN {X 0,Y 608.543,Z 537.44,A -85,B 0,C 180,E1 -461.597,E2 -461.597} C_VEL
LIN {X 0,Y 608.443,Z 527.53,A -85,B 0,C 180,E1 -461.789,E2 -461.789} C_VEL
LIN {X 0,Y 608.442,Z 517.436,A -85,B 0,C 180,E1 -464.379,E2 -464.379} C_VEL
LIN {X 0,Y 608.447,Z 506.844,A -85,B 0,C 180,E1 -467.13,E2 -467.13} C_VEL
LIN {X 0,Y 608.453,Z 496.253,A -85,B 0,C 180,E1 -469.922,E2 -469.922} C_VEL
LIN {X 0,Y 608.462,Z 485.663,A -85,B 0,C 180,E1 -472.764,E2 -472.764} C_VEL
LIN {X 0,Y 608.469,Z 476.395,A -85,B 0,C 180,E1 -475.3,E2 -475.3} C_VEL
LIN {X 0,Y 608.497,Z 467.127,A -85,B 0,C 180,E1 -477.889,E2 -477.889} C_VEL
LIN {X 0,Y 608.538,Z 457.86,A -85,B 0,C 180,E1 -480.541,E2 -480.541} C_VEL
LIN {X 0,Y 608.527,Z 448.583,A -85,B 0,C 180,E1 -483.27,E2 -483.27} C_VEL
LIN {X 0,Y 608.482,Z 440.689,A -85,B 0,C 180,E1 -485.704,E2 -485.704} C_VEL
LIN {X 0,Y 608.47,Z 440.692,A -85,B 0,C 180,E1 -488.588,E2 -488.588} C_VEL
LIN {X 0,Y 608.467,Z 440.696,A -85,B 0,C 180,E1 -491.343,E2 -491.343} C_VEL
LIN {X 0,Y 608.451,Z 440.695,A -85,B 0,C 180,E1 -494.263,E2 -494.263} C_VEL
LIN {X 0,Y 608.455,Z 440.692,A -85,B 0,C 180,E1 -497.04,E2 -497.04} C_VEL
LIN {X 0,Y 608.454,Z 440.692,A -85,B 0,C 180,E1 -499.697,E2 -499.697} C_VEL
LIN {X 0,Y 608.47,Z 440.695,A -85,B 0,C 180,E1 -502.254,E2 -502.254} C_VEL
LIN {X 0,Y 608.452,Z 440.694,A -85,B 0,C 180,E1 -505.094,E2 -505.094} C_VEL
LIN {X 0,Y 608.47,Z 440.689,A -85,B 0,C 180,E1 -507.906,E2 -507.906} C_VEL
LIN {X 0,Y 608.481,Z 440.693,A -85,B 0,C 180,E1 -510.221,E2 -510.221} C_VEL
LIN {X 0,Y 608.457,Z 440.697,A -85,B 0,C 180,E1 -513.226,E2 -513.226} C_VEL
LIN {X 0,Y 608.466,Z 440.693,A -85,B 0,C 180,E1 -516.155,E2 -516.155} C_VEL
LIN {X 0,Y 608.478,Z 440.69,A -85,B 0,C 180,E1 -518.309,E2 -518.309} C_VEL
LIN {X 0,Y 608.473,Z 440.692,A -85,B 0,C 180,E1 -521.284,E2 -521.284} C_VEL
LIN {X 0,Y 608.461,Z 440.693,A -85,B 0,C 180,E1 -523.906,E2 -523.906} C_VEL
LIN {X 0,Y 608.466,Z 440.69,A -85,B 0,C 180,E1 -526.644,E2 -526.644} C_VEL
LIN {X 0,Y 608.468,Z 440.69,A -85,B 0,C 180,E1 -529.35,E2 -529.35} C_VEL
LIN {X 0,Y 608.484,Z 440.694,A -85,B 0,C 180,E1 -532.033,E2 -532.033} C_VEL
LIN {X 0,Y 608.47,Z 440.691,A -85,B 0,C 180,E1 -534.698,E2 -534.698} C_VEL
LIN {X 0,Y 608.48,Z 440.688,A -85,B 0,C 180,E1 -537.352,E2 -537.352} C_VEL
LIN {X 0,Y 608.48,Z 440.692,A -85,B 0,C 180,E1 -540,E2 -540} C_VEL
LIN {X 0,Y 608.487,Z 440.691,A -85,B 0,C 180,E1 -542.648,E2 -542.648} C_VEL
LIN {X 0,Y 608.464,Z 440.69,A -85,B 0,C 180,E1 -545.302,E2 -545.302} C_VEL
LIN {X 0,Y 608.477,Z 440.69,A -85,B 0,C 180,E1 -547.967,E2 -547.967} C_VEL
LIN {X 0,Y 608.457,Z 440.693,A -85,B 0,C 180,E1 -549.459,E2 -549.459} C_VEL
LIN {X 0,Y 607.775,Z 440.776,A -85,B 0,C 180,E1 -550.012,E2 -550.012} C_VEL
LIN {X 0,Y 604.92,Z 441.135,A -85,B 0,C 180,E1 -550.909,E2 -550.909} C_VEL
LIN {X 0,Y 602.519,Z 441.436,A -85,B 0,C 180,E1 -551.63,E2 -551.63} C_VEL
LIN {X 0,Y 601.491,Z 441.564,A -85,B 0,C 180,E1 -552.187,E2 -552.187} C_VEL
LIN {X 0,Y 601.408,Z 441.571,A -85,B 0,C 180,E1 -552.376,E2 -552.376} C_VEL
LIN {X 0,Y 601.432,Z 441.567,A -85,B 0,C 180,E1 -554.897,E2 -554.897} C_VEL
LIN {X 0,Y 601.436,Z 441.571,A -85,B 0,C 180,E1 -556.986,E2 -556.986} C_VEL
LIN {X 0,Y 601.409,Z 441.572,A -85,B 0,C 180,E1 -559.81,E2 -559.81} C_VEL
LIN {X 0,Y 601.415,Z 441.569,A -85,B 0,C 180,E1 -562.683,E2 -562.683} C_VEL
LIN {X 0,Y 601.403,Z 441.574,A -85,B 0,C 180,E1 -564.879,E2 -564.879} C_VEL
LIN {X 0,Y 601.423,Z 441.574,A -85,B 0,C 180,E1 -567.868,E2 -567.868} C_VEL
LIN {X 0,Y 601.431,Z 441.566,A -85,B 0,C 180,E1 -570.164,E2 -570.164} C_VEL
LIN {X 0,Y 601.429,Z 441.57,A -85,B 0,C 180,E1 -572.716,E2 -572.716} C_VEL
LIN {X 0,Y 601.397,Z 441.571,A -85,B 0,C 180,E1 -575.112,E2 -575.112} C_VEL
LIN {X 0,Y 601.438,Z 441.569,A -85,B 0,C 180,E1 -577.419,E2 -577.419} C_VEL
LIN {X 0,Y 601.404,Z 441.572,A -85,B 0,C 180,E1 -579.996,E2 -579.996} C_VEL
LIN {X 0,Y 601.415,Z 441.568,A -85,B 0,C 180,E1 -582.67,E2 -582.67} C_VEL
LIN {X 0,Y 601.43,Z 441.567,A -85,B 0,C 180,E1 -585.482,E2 -585.482} C_VEL
LIN {X 0,Y 601.423,Z 441.57,A -85,B 0,C 180,E1 -588.408,E2 -588.408} C_VEL
LIN {X 0,Y 601.416,Z 441.57,A -85,B 0,C 180,E1 -590.874,E2 -590.874} C_VEL
LIN {X 0,Y 601.403,Z 441.57,A -85,B 0,C 180,E1 -593.417,E2 -593.417} C_VEL
LIN {X 0,Y 601.437,Z 441.57,A -85,B 0,C 180,E1 -596.064,E2 -596.064} C_VEL
LIN {X 0,Y 601.425,Z 441.568,A -85,B 0,C 180,E1 -598.545,E2 -598.545} C_VEL
LIN {X 0,Y 601.43,Z 441.566,A -85,B 0,C 180,E1 -601.373,E2 -601.373} C_VEL
LIN {X 0,Y 601.404,Z 441.575,A -85,B 0,C 180,E1 -603.636,E2 -603.636} C_VEL
LIN {X 0,Y 601.423,Z 441.57,A -85,B 0,C 180,E1 -606.59,E2 -606.59} C_VEL
LIN {X 0,Y 601.43,Z 441.567,A -85,B 0,C 180,E1 -609.478,E2 -609.478} C_VEL
LIN {X 0,Y 601.399,Z 441.57,A -85,B 0,C 180,E1 -612.312,E2 -612.312} C_VEL
LIN {X 0,Y 601.416,Z 441.571,A -85,B 0,C 180,E1 -614.409,E2 -614.409} C_VEL
LIN {X 0,Y 601.418,Z 441.568,A -85,B 0,C 180,E1 -617.172,E2 -617.172} C_VEL
LIN {X 0,Y 601.439,Z 441.566,A -85,B 0,C 180,E1 -619.905,E2 -619.905} C_VEL
LIN {X 0,Y 601.445,Z 441.569,A -85,B 0,C 180,E1 -622.615,E2 -622.615} C_VEL
LIN {X 0,Y 601.421,Z 441.57,A -85,B 0,C 180,E1 -625.308,E2 -625.308} C_VEL
LIN {X 0,Y 601.437,Z 441.566,A -85,B 0,C 180,E1 -627.991,E2 -627.991} C_VEL
LIN {X 0,Y 601.447,Z 441.565,A -85,B 0,C 180,E1 -630.67,E2 -630.67} C_VEL
LIN {X 0,Y 601.432,Z 441.573,A -85,B 0,C 180,E1 -633.35,E2 -633.35} C_VEL
LIN {X 0,Y 601.42,Z 441.569,A -85,B 0,C 180,E1 -636.037,E2 -636.037} C_VEL
LIN {X 0,Y 601.414,Z 441.568,A -85,B 0,C 180,E1 -638.738,E2 -638.738} C_VEL
LIN {X 0,Y 601.443,Z 441.567,A -85,B 0,C 180,E1 -641.458,E2 -641.458} C_VEL
LIN {X 0,Y 601.425,Z 441.573,A -85,B 0,C 180,E1 -644.205,E2 -644.205} C_VEL
LIN {X 0,Y 601.418,Z 441.569,A -85,B 0,C 180,E1 -646.986,E2 -646.986} C_VEL
LIN {X 0,Y 601.408,Z 441.569,A -85,B 0,C 180,E1 -649.81,E2 -649.81} C_VEL
LIN {X 0,Y 601.422,Z 441.568,A -85,B 0,C 180,E1 -652.606,E2 -652.606} C_VEL
LIN {X 0,Y 601.405,Z 441.572,A -85,B 0,C 180,E1 -654.879,E2 -654.879} C_VEL
LIN {X 0,Y 601.416,Z 441.568,A -85,B 0,C 180,E1 -657.362,E2 -657.362} C_VEL
LIN {X 0,Y 601.434,Z 441.569,A -85,B 0,C 180,E1 -660.164,E2 -660.164} C_VEL
LIN {X 0,Y 601.419,Z 441.57,A -85,B 0,C 180,E1 -662.714,E2 -662.714} C_VEL
LIN {X 0,Y 601.405,Z 441.57,A -85,B 0,C 180,E1 -665.113,E2 -665.113} C_VEL
LIN {X 0,Y 601.438,Z 441.568,A -85,B 0,C 180,E1 -667.419,E2 -667.419} C_VEL
LIN {X 0,Y 601.416,Z 441.568,A -85,B 0,C 180,E1 -669.995,E2 -669.995} C_VEL
LIN {X 0,Y 601.416,Z 441.571,A -85,B 0,C 180,E1 -672.67,E2 -672.67} C_VEL
LIN {X 0,Y 601.431,Z 441.573,A -85,B 0,C 180,E1 -675.482,E2 -675.482} C_VEL
LIN {X 0,Y 601.428,Z 441.571,A -85,B 0,C 180,E1 -678.407,E2 -678.407} C_VEL
LIN {X 0,Y 601.408,Z 441.569,A -85,B 0,C 180,E1 -680.873,E2 -680.873} C_VEL
LIN {X 0,Y 601.406,Z 441.574,A -85,B 0,C 180,E1 -683.417,E2 -683.417} C_VEL
LIN {X 0,Y 601.353,Z 441.581,A -85,B 0,C 180,E1 -685.064,E2 -685.064} C_VEL
LIN {X 0,Y 601.372,Z 444.405,A -85,B 0,C 180,E1 -687.48,E2 -687.48} C_VEL
LIN {X 0,Y 601.362,Z 447.239,A -85,B 0,C 180,E1 -689.863,E2 -689.863} C_VEL
LIN {X 0,Y 601.346,Z 450.743,A -85,B 0,C 180,E1 -692.651,E2 -692.651} C_VEL
LIN {X 0,Y 601.344,Z 453.921,A -85,B 0,C 180,E1 -695.119,E2 -695.119} C_VEL
LIN {X 0,Y 601.339,Z 457.765,A -85,B 0,C 180,E1 -698.038,E2 -698.038} C_VEL
LIN {X 0,Y 601.315,Z 460.647,A -85,B 0,C 180,E1 -700.187,E2 -700.187} C_VEL
LIN {X 0,Y 601.338,Z 464.49,A -85,B 0,C 180,E1 -703.011,E2 -703.011} C_VEL
LIN {X 0,Y 601.338,Z 468.541,A -85,B 0,C 180,E1 -705.941,E2 -705.941} C_VEL
LIN {X 0,Y 601.337,Z 471.667,A -85,B 0,C 180,E1 -708.177,E2 -708.177} C_VEL
LIN {X 0,Y 601.584,Z 477.332,A -85,B 0,C 180,E1 -708.31,E2 -708.31} C_VEL
LIN {X 0,Y 601.567,Z 490.86,A -85,B 0,C 180,E1 -708.688,E2 -708.688} C_VEL
LIN {X 0,Y 601.549,Z 503.099,A -85,B 0,C 180,E1 -709.171,E2 -709.171} C_VEL
LIN {X 0,Y 601.492,Z 515.419,A -85,B 0,C 180,E1 -709.821,E2 -709.821} C_VEL
LIN {X 0,Y 601.455,Z 526.796,A -85,B 0,C 180,E1 -710.585,E2 -710.585} C_VEL
LIN {X 0,Y 601.424,Z 536.863,A -85,B 0,C 180,E1 -711.431,E2 -711.431} C_VEL
LIN {X 0,Y 601.418,Z 546.567,A -85,B 0,C 180,E1 -712.446,E2 -712.446} C_VEL
LIN {X 0,Y 601.377,Z 553.888,A -85,B 0,C 180,E1 -713.393,E2 -713.393} C_VEL
LIN {X 0,Y 601.372,Z 559.612,A -85,B 0,C 180,E1 -714.299,E2 -714.299} C_VEL
LIN {X 0,Y 601.335,Z 564.753,A -85,B 0,C 180,E1 -715.307,E2 -715.307} C_VEL
LIN {X 0,Y 601.368,Z 568.743,A -85,B 0,C 180,E1 -716.315,E2 -716.315} C_VEL
LIN {X 0,Y 601.325,Z 571.692,A -85,B 0,C 180,E1 -717.32,E2 -717.32} C_VEL
LIN {X 0,Y 601.341,Z 573.127,A -85,B 0,C 180,E1 -717.991,E2 -717.991} C_VEL
LIN {X 0,Y 601.34,Z 574.752,A -85,B 0,C 180,E1 -719.33,E2 -719.33} C_VEL
LIN {X 0,Y 601.335,Z 574.996,A -85,B 0,C 180,E1 -720,E2 -720} C_VEL
LIN {X 0,Y 601.339,Z 574.815,A -85,B 0,C 180,E1 -720.67,E2 -720.67} C_VEL
LIN {X 0,Y 601.34,Z 573.276,A -85,B 0,C 180,E1 -722.009,E2 -722.009} C_VEL
LIN {X 0,Y 601.326,Z 571.917,A -85,B 0,C 180,E1 -722.679,E2 -722.679} C_VEL
LIN {X 0,Y 601.369,Z 569.04,A -85,B 0,C 180,E1 -723.685,E2 -723.685} C_VEL
LIN {X 0,Y 601.337,Z 565.141,A -85,B 0,C 180,E1 -724.693,E2 -724.693} C_VEL
LIN {X 0,Y 601.373,Z 560.11,A -85,B 0,C 180,E1 -725.701,E2 -725.701} C_VEL
LIN {X 0,Y 601.382,Z 553.792,A -85,B 0,C 180,E1 -726.711,E2 -726.711} C_VEL
LIN {X 0,Y 601.396,Z 545.875,A -85,B 0,C 180,E1 -727.723,E2 -727.723} C_VEL
LIN {X 0,Y 601.436,Z 536.031,A -85,B 0,C 180,E1 -728.738,E2 -728.738} C_VEL
LIN {X 0,Y 601.446,Z 525.709,A -85,B 0,C 180,E1 -729.585,E2 -729.585} C_VEL
LIN {X 0,Y 601.493,Z 514.09,A -85,B 0,C 180,E1 -730.349,E2 -730.349} C_VEL
LIN {X 0,Y 601.531,Z 502.077,A -85,B 0,C 180,E1 -730.964,E2 -730.964} C_VEL
LIN {X 0,Y 601.552,Z 489.247,A -85,B 0,C 180,E1 -731.456,E2 -731.456} C_VEL
LIN {X 0,Y 601.579,Z 476.623,A -85,B 0,C 180,E1 -731.797,E2 -731.797} C_VEL
LIN {X 0,Y 601.334,Z 471.673,A -85,B 0,C 180,E1 -731.909,E2 -731.909} C_VEL
LIN {X 0,Y 601.319,Z 468.459,A -85,B 0,C 180,E1 -734.208,E2 -734.208} C_VEL
LIN {X 0,Y 601.338,Z 464.614,A -85,B 0,C 180,E1 -736.989,E2 -736.989} C_VEL
LIN {X 0,Y 601.315,Z 460.769,A -85,B 0,C 180,E1 -739.813,E2 -739.813} C_VEL
LIN {X 0,Y 601.338,Z 457.885,A -85,B 0,C 180,E1 -741.962,E2 -741.962} C_VEL
LIN {X 0,Y 601.345,Z 454.039,A -85,B 0,C 180,E1 -744.881,E2 -744.881} C_VEL
LIN {X 0,Y 601.344,Z 450.858,A -85,B 0,C 180,E1 -747.349,E2 -747.349} C_VEL
LIN {X 0,Y 601.359,Z 447.318,A -85,B 0,C 180,E1 -750.168,E2 -750.168} C_VEL
LIN {X 0,Y 601.381,Z 444.549,A -85,B 0,C 180,E1 -752.709,E2 -752.709} C_VEL
LIN {X 0,Y 601.389,Z 441.787,A -85,B 0,C 180,E1 -755.111,E2 -755.111} C_VEL
LIN {X 0,Y 601.439,Z 441.569,A -85,B 0,C 180,E1 -757.419,E2 -757.419} C_VEL
LIN {X 0,Y 601.405,Z 441.574,A -85,B 0,C 180,E1 -759.996,E2 -759.996} C_VEL
LIN {X 0,Y 601.417,Z 441.575,A -85,B 0,C 180,E1 -762.67,E2 -762.67} C_VEL
LIN {X 0,Y 601.43,Z 441.57,A -85,B 0,C 180,E1 -765.482,E2 -765.482} C_VEL
LIN {X 0,Y 601.427,Z 441.571,A -85,B 0,C 180,E1 -768.407,E2 -768.407} C_VEL
LIN {X 0,Y 601.438,Z 441.57,A -85,B 0,C 180,E1 -770.875,E2 -770.875} C_VEL
LIN {X 0,Y 601.404,Z 441.576,A -85,B 0,C 180,E1 -773.417,E2 -773.417} C_VEL
LIN {X 0,Y 601.443,Z 441.695,A -85,B 0,C 180,E1 -774.024,E2 -774.024} C_VEL
LIN {X 0,Y 601.602,Z 445.994,A -85,B 0,C 180,E1 -775.487,E2 -775.487} C_VEL
LIN {X 0,Y 601.558,Z 453.803,A -85,B 0,C 180,E1 -777.888,E2 -777.888} C_VEL
LIN {X 0,Y 601.521,Z 463.155,A -85,B 0,C 180,E1 -780.612,E2 -780.612} C_VEL
LIN {X 0,Y 601.512,Z 472.422,A -85,B 0,C 180,E1 -783.267,E2 -783.267} C_VEL
LIN {X 0,Y 601.46,Z 483.013,A -85,B 0,C 180,E1 -786.226,E2 -786.226} C_VEL
LIN {X 0,Y 601.442,Z 492.281,A -85,B 0,C 180,E1 -788.762,E2 -788.762} C_VEL
LIN {X 0,Y 601.401,Z 502.872,A -85,B 0,C 180,E1 -791.607,E2 -791.607} C_VEL
LIN {X 0,Y 601.385,Z 513.463,A -85,B 0,C 180,E1 -794.408,E2 -794.408} C_VEL
LIN {X 0,Y 601.362,Z 524.054,A -85,B 0,C 180,E1 -797.17,E2 -797.17} C_VEL
LIN {X 0,Y 601.387,Z 527.53,A -85,B 0,C 180,E1 -798.071,E2 -798.071} C_VEL
LIN {X 0,Y 601.601,Z 540.176,A -85,B 0,C 180,E1 -798.331,E2 -798.331} C_VEL
LIN {X 0,Y 601.568,Z 552.203,A -85,B 0,C 180,E1 -798.687,E2 -798.687} C_VEL
LIN {X 0,Y 601.511,Z 564.016,A -85,B 0,C 180,E1 -799.169,E2 -799.169} C_VEL
LIN {X 0,Y 601.494,Z 576.166,A -85,B 0,C 180,E1 -799.821,E2 -799.821} C_VEL
LIN {X 0,Y 601.455,Z 587.401,A -85,B 0,C 180,E1 -800.585,E2 -800.585} C_VEL
LIN {X 0,Y 601.423,Z 597.335,A -85,B 0,C 180,E1 -801.431,E2 -801.431} C_VEL
LIN {X 0,Y 601.418,Z 606.959,A -85,B 0,C 180,E1 -802.446,E2 -802.446} C_VEL
LIN {X 0,Y 601.37,Z 614.224,A -85,B 0,C 180,E1 -803.398,E2 -803.398} C_VEL
LIN {X 0,Y 601.372,Z 619.865,A -85,B 0,C 180,E1 -804.299,E2 -804.299} C_VEL
LIN {X 0,Y 601.337,Z 624.95,A -85,B 0,C 180,E1 -805.307,E2 -805.307} C_VEL
LIN {X 0,Y 601.367,Z 628.896,A -85,B 0,C 180,E1 -806.315,E2 -806.315} C_VEL
LIN {X 0,Y 601.325,Z 631.809,A -85,B 0,C 180,E1 -807.32,E2 -807.32} C_VEL
LIN {X 0,Y 601.341,Z 633.201,A -85,B 0,C 180,E1 -807.991,E2 -807.991} C_VEL
LIN {X 0,Y 601.339,Z 634.784,A -85,B 0,C 180,E1 -809.33,E2 -809.33} C_VEL
LIN {X 0,Y 601.335,Z 635,A -85,B 0,C 180,E1 -810,E2 -810} C_VEL
LIN {X 0,Y 601.348,Z 634.184,A -85,B 0,C 180,E1 -811.339,E2 -811.339} C_VEL
LIN {X 0,Y 601.341,Z 633.202,A -85,B 0,C 180,E1 -812.009,E2 -812.009} C_VEL
LIN {X 0,Y 601.325,Z 631.809,A -85,B 0,C 180,E1 -812.679,E2 -812.679} C_VEL
LIN {X 0,Y 601.367,Z 628.896,A -85,B 0,C 180,E1 -813.685,E2 -813.685} C_VEL
LIN {X 0,Y 601.337,Z 624.95,A -85,B 0,C 180,E1 -814.693,E2 -814.693} C_VEL
LIN {X 0,Y 601.372,Z 618.877,A -85,B 0,C 180,E1 -815.869,E2 -815.869} C_VEL
LIN {X 0,Y 601.382,Z 612.236,A -85,B 0,C 180,E1 -816.88,E2 -816.88} C_VEL
LIN {X 0,Y 601.4,Z 603.99,A -85,B 0,C 180,E1 -817.892,E2 -817.892} C_VEL
LIN {X 0,Y 601.436,Z 595.537,A -85,B 0,C 180,E1 -818.738,E2 -818.738} C_VEL
LIN {X 0,Y 601.449,Z 585.092,A -85,B 0,C 180,E1 -819.585,E2 -819.585} C_VEL
LIN {X 0,Y 601.472,Z 574.757,A -85,B 0,C 180,E1 -820.264,E2 -820.264} C_VEL
LIN {X 0,Y 601.534,Z 562.637,A -85,B 0,C 180,E1 -820.894,E2 -820.894} C_VEL
LIN {X 0,Y 601.568,Z 550.225,A -85,B 0,C 180,E1 -821.378,E2 -821.378} C_VEL
LIN {X 0,Y 601.599,Z 537.439,A -85,B 0,C 180,E1 -821.732,E2 -821.732} C_VEL
LIN {X 0,Y 601.387,Z 527.53,A -85,B 0,C 180,E1 -821.929,E2 -821.929} C_VEL
LIN {X 0,Y 601.39,Z 517.436,A -85,B 0,C 180,E1 -824.552,E2 -824.552} C_VEL
LIN {X 0,Y 601.389,Z 506.844,A -85,B 0,C 180,E1 -827.338,E2 -827.338} C_VEL
LIN {X 0,Y 601.424,Z 496.253,A -85,B 0,C 180,E1 -830.165,E2 -830.165} C_VEL
LIN {X 0,Y 601.431,Z 485.662,A -85,B 0,C 180,E1 -833.046,E2 -833.046} C_VEL
LIN {X 0,Y 601.471,Z 476.395,A -85,B 0,C 180,E1 -835.616,E2 -835.616} C_VEL
LIN {X 0,Y 601.495,Z 467.127,A -85,B 0,C 180,E1 -838.243,E2 -838.243} C_VEL
LIN {X 0,Y 601.543,Z 457.86,A -85,B 0,C 180,E1 -840.935,E2 -840.935} C_VEL
LIN {X 0,Y 601.584,Z 449.884,A -85,B 0,C 180,E1 -843.304,E2 -843.304} C_VEL
LIN {X 0,Y 601.598,Z 443.941,A -85,B 0,C 180,E1 -845.139,E2 -845.139} C_VEL
LIN {X 0,Y 601.433,Z 441.568,A -85,B 0,C 180,E1 -845.932,E2 -845.932} C_VEL
LIN {X 0,Y 601.435,Z 441.57,A -85,B 0,C 180,E1 -848.471,E2 -848.471} C_VEL
LIN {X 0,Y 601.419,Z 441.569,A -85,B 0,C 180,E1 -850.874,E2 -850.874} C_VEL
LIN {X 0,Y 601.43,Z 441.567,A -85,B 0,C 180,E1 -853.586,E2 -853.586} C_VEL
LIN {X 0,Y 601.453,Z 441.566,A -85,B 0,C 180,E1 -856.425,E2 -856.425} C_VEL
LIN {X 0,Y 601.417,Z 441.572,A -85,B 0,C 180,E1 -859.427,E2 -859.427} C_VEL
LIN {X 0,Y 601.418,Z 441.568,A -85,B 0,C 180,E1 -861.732,E2 -861.732} C_VEL
LIN {X 0,Y 601.39,Z 441.573,A -85,B 0,C 180,E1 -864.245,E2 -864.245} C_VEL
LIN {X 0,Y 601.423,Z 441.57,A -85,B 0,C 180,E1 -866.686,E2 -866.686} C_VEL
LIN {X 0,Y 601.414,Z 441.569,A -85,B 0,C 180,E1 -869.058,E2 -869.058} C_VEL
LIN {X 0,Y 601.433,Z 441.568,A -85,B 0,C 180,E1 -871.373,E2 -871.373} C_VEL
LIN {X 0,Y 601.407,Z 441.571,A -85,B 0,C 180,E1 -873.636,E2 -873.636} C_VEL
LIN {X 0,Y 601.419,Z 441.571,A -85,B 0,C 180,E1 -876.59,E2 -876.59} C_VEL
LIN {X 0,Y 601.433,Z 441.573,A -85,B 0,C 180,E1 -879.478,E2 -879.478} C_VEL
LIN {X 0,Y 601.396,Z 441.573,A -85,B 0,C 180,E1 -882.312,E2 -882.312} C_VEL
LIN {X 0,Y 601.415,Z 441.572,A -85,B 0,C 180,E1 -884.409,E2 -884.409} C_VEL
LIN {X 0,Y 601.424,Z 441.572,A -85,B 0,C 180,E1 -887.172,E2 -887.172} C_VEL
LIN {X 0,Y 601.431,Z 441.567,A -85,B 0,C 180,E1 -889.905,E2 -889.905} C_VEL
LIN {X 0,Y 601.443,Z 441.565,A -85,B 0,C 180,E1 -892.615,E2 -892.615} C_VEL
LIN {X 0,Y 601.428,Z 441.57,A -85,B 0,C 180,E1 -895.308,E2 -895.308} C_VEL
LIN {X 0,Y 601.423,Z 441.571,A -85,B 0,C 180,E1 -897.991,E2 -897.991} C_VEL
LIN {X 0,Y 601.454,Z 441.564,A -85,B 0,C 180,E1 -900.67,E2 -900.67} C_VEL
LIN {X 0,Y 601.429,Z 441.568,A -85,B 0,C 180,E1 -903.35,E2 -903.35} C_VEL
LIN {X 0,Y 601.413,Z 441.575,A -85,B 0,C 180,E1 -906.037,E2 -906.037} C_VEL
LIN {X 0,Y 601.439,Z 441.567,A -85,B 0,C 180,E1 -908.738,E2 -908.738} C_VEL
LIN {X 0,Y 601.424,Z 441.567,A -85,B 0,C 180,E1 -911.459,E2 -911.459} C_VEL
LIN {X 0,Y 601.408,Z 441.571,A -85,B 0,C 180,E1 -912.376,E2 -912.376} C_VEL
LIN {X 0,Y 600.746,Z 441.653,A -85,B 0,C 180,E1 -912.935,E2 -912.935} C_VEL
LIN {X 0,Y 597.897,Z 442.013,A -85,B 0,C 180,E1 -913.843,E2 -913.843} C_VEL
LIN {X 0,Y 595.487,Z 442.312,A -85,B 0,C 180,E1 -914.573,E2 -914.573} C_VEL
LIN {X 0,Y 594.448,Z 442.44,A -85,B 0,C 180,E1 -915.137,E2 -915.137} C_VEL
LIN {X 0,Y 594.362,Z 442.448,A -85,B 0,C 180,E1 -915.327,E2 -915.327} C_VEL
LIN {X 0,Y 594.392,Z 442.446,A -85,B 0,C 180,E1 -917.193,E2 -917.193} C_VEL
LIN {X 0,Y 594.378,Z 442.451,A -85,B 0,C 180,E1 -920.054,E2 -920.054} C_VEL
LIN {X 0,Y 594.366,Z 442.45,A -85,B 0,C 180,E1 -922.967,E2 -922.967} C_VEL
LIN {X 0,Y 594.376,Z 442.446,A -85,B 0,C 180,E1 -925.193,E2 -925.193} C_VEL
LIN {X 0,Y 594.389,Z 442.446,A -85,B 0,C 180,E1 -927.527,E2 -927.527} C_VEL
LIN {X 0,Y 594.389,Z 442.444,A -85,B 0,C 180,E1 -930.328,E2 -930.328} C_VEL
LIN {X 0,Y 594.383,Z 442.445,A -85,B 0,C 180,E1 -932.95,E2 -932.95} C_VEL
LIN {X 0,Y 594.359,Z 442.45,A -85,B 0,C 180,E1 -935.409,E2 -935.409} C_VEL
LIN {X 0,Y 594.388,Z 442.444,A -85,B 0,C 180,E1 -937.941,E2 -937.941} C_VEL
LIN {X 0,Y 594.377,Z 442.446,A -85,B 0,C 180,E1 -940.822,E2 -940.822} C_VEL
LIN {X 0,Y 594.387,Z 442.446,A -85,B 0,C 180,E1 -943.841,E2 -943.841} C_VEL
LIN {X 0,Y 594.369,Z 442.451,A -85,B 0,C 180,E1 -946.701,E2 -946.701} C_VEL
LIN {X 0,Y 594.372,Z 442.449,A -85,B 0,C 180,E1 -949.433,E2 -949.433} C_VEL
LIN {X 0,Y 594.393,Z 442.444,A -85,B 0,C 180,E1 -952.392,E2 -952.392} C_VEL
LIN {X 0,Y 594.402,Z 442.442,A -85,B 0,C 180,E1 -955.421,E2 -955.421} C_VEL
LIN {X 0,Y 594.383,Z 442.444,A -85,B 0,C 180,E1 -958.357,E2 -958.357} C_VEL
LIN {X 0,Y 594.387,Z 442.445,A -85,B 0,C 180,E1 -961.042,E2 -961.042} C_VEL
LIN {X 0,Y 594.388,Z 442.447,A -85,B 0,C 180,E1 -963.978,E2 -963.978} C_VEL
LIN {X 0,Y 594.392,Z 442.444,A -85,B 0,C 180,E1 -966.296,E2 -966.296} C_VEL
LIN {X 0,Y 594.405,Z 442.441,A -85,B 0,C 180,E1 -969.224,E2 -969.224} C_VEL
LIN {X 0,Y 594.358,Z 442.448,A -85,B 0,C 180,E1 -972.095,E2 -972.095} C_VEL
LIN {X 0,Y 594.369,Z 442.447,A -85,B 0,C 180,E1 -974.219,E2 -974.219} C_VEL
LIN {X 0,Y 594.386,Z 442.449,A -85,B 0,C 180,E1 -976.321,E2 -976.321} C_VEL
LIN {X 0,Y 594.381,Z 442.448,A -85,B 0,C 180,E1 -979.095,E2 -979.095} C_VEL
LIN {X 0,Y 594.418,Z 442.44,A -85,B 0,C 180,E1 -981.843,E2 -981.843} C_VEL
LIN {X 0,Y 594.392,Z 442.443,A -85,B 0,C 180,E1 -984.572,E2 -984.572} C_VEL
LIN {X 0,Y 594.408,Z 442.445,A -85,B 0,C 180,E1 -987.289,E2 -987.289} C_VEL
LIN {X 0,Y 594.42,Z 442.443,A -85,B 0,C 180,E1 -990,E2 -990} C_VEL
LIN {X 0,Y 594.405,Z 442.442,A -85,B 0,C 180,E1 -992.711,E2 -992.711} C_VEL
LIN {X 0,Y 594.393,Z 442.444,A -85,B 0,C 180,E1 -995.428,E2 -995.428} C_VEL
LIN {X 0,Y 594.397,Z 442.443,A -85,B 0,C 180,E1 -997.473,E2 -997.473} C_VEL
LIN {X 0,Y 594.397,Z 442.443,A -85,B 0,C 180,E1 -1000.216,E2 -1000.216} C_VEL
LIN {X 0,Y 594.368,Z 442.449,A -85,B 0,C 180,E1 -1002.983,E2 -1002.983} C_VEL
LIN {X 0,Y 594.372,Z 442.445,A -85,B 0,C 180,E1 -1005.078,E2 -1005.078} C_VEL
LIN {X 0,Y 594.384,Z 442.448,A -85,B 0,C 180,E1 -1007.194,E2 -1007.194} C_VEL
LIN {X 0,Y 594.379,Z 442.446,A -85,B 0,C 180,E1 -1010.054,E2 -1010.054} C_VEL
LIN {X 0,Y 594.369,Z 442.446,A -85,B 0,C 180,E1 -1012.967,E2 -1012.967} C_VEL
LIN {X 0,Y 594.38,Z 442.451,A -85,B 0,C 180,E1 -1015.193,E2 -1015.193} C_VEL
LIN {X 0,Y 594.373,Z 442.445,A -85,B 0,C 180,E1 -1017.523,E2 -1017.523} C_VEL
LIN {X 0,Y 594.391,Z 442.444,A -85,B 0,C 180,E1 -1020.328,E2 -1020.328} C_VEL
LIN {X 0,Y 594.381,Z 442.451,A -85,B 0,C 180,E1 -1022.95,E2 -1022.95} C_VEL
LIN {X 0,Y 594.357,Z 442.447,A -85,B 0,C 180,E1 -1025.409,E2 -1025.409} C_VEL
LIN {X 0,Y 594.386,Z 442.447,A -85,B 0,C 180,E1 -1027.941,E2 -1027.941} C_VEL
LIN {X 0,Y 594.375,Z 442.451,A -85,B 0,C 180,E1 -1030.821,E2 -1030.821} C_VEL
LIN {X 0,Y 594.371,Z 442.446,A -85,B 0,C 180,E1 -1033.299,E2 -1033.299} C_VEL
LIN {X 0,Y 594.373,Z 442.446,A -85,B 0,C 180,E1 -1036.16,E2 -1036.16} C_VEL
LIN {X 0,Y 594.385,Z 442.45,A -85,B 0,C 180,E1 -1038.536,E2 -1038.536} C_VEL
LIN {X 0,Y 594.377,Z 442.446,A -85,B 0,C 180,E1 -1041.297,E2 -1041.297} C_VEL
LIN {X 0,Y 594.356,Z 442.449,A -85,B 0,C 180,E1 -1043.755,E2 -1043.755} C_VEL
LIN {X 0,Y 594.294,Z 442.551,A -85,B 0,C 180,E1 -1045.414,E2 -1045.414} C_VEL
LIN {X 0,Y 594.307,Z 446.033,A -85,B 0,C 180,E1 -1048.369,E2 -1048.369} C_VEL
LIN {X 0,Y 594.259,Z 449.209,A -85,B 0,C 180,E1 -1051.065,E2 -1051.065} C_VEL
LIN {X 0,Y 594.259,Z 452.001,A -85,B 0,C 180,E1 -1053.294,E2 -1053.294} C_VEL
LIN {X 0,Y 594.281,Z 454.936,A -85,B 0,C 180,E1 -1055.59,E2 -1055.59} C_VEL
LIN {X 0,Y 594.225,Z 458.726,A -85,B 0,C 180,E1 -1058.491,E2 -1058.491} C_VEL
LIN {X 0,Y 594.243,Z 462.212,A -85,B 0,C 180,E1 -1061.111,E2 -1061.111} C_VEL
LIN {X 0,Y 594.249,Z 465.452,A -85,B 0,C 180,E1 -1063.51,E2 -1063.51} C_VEL
LIN {X 0,Y 594.247,Z 469.295,A -85,B 0,C 180,E1 -1066.318,E2 -1066.318} C_VEL
LIN {X 0,Y 594.263,Z 471.668,A -85,B 0,C 180,E1 -1068.034,E2 -1068.034} C_VEL
LIN {X 0,Y 594.647,Z 476.439,A -85,B 0,C 180,E1 -1068.15,E2 -1068.15} C_VEL
LIN {X 0,Y 594.621,Z 489.104,A -85,B 0,C 180,E1 -1068.495,E2 -1068.495} C_VEL
LIN {X 0,Y 594.535,Z 501.545,A -85,B 0,C 180,E1 -1068.973,E2 -1068.973} C_VEL
LIN {X 0,Y 594.502,Z 512.521,A -85,B 0,C 180,E1 -1069.528,E2 -1069.528} C_VEL
LIN {X 0,Y 594.449,Z 523.314,A -85,B 0,C 180,E1 -1070.215,E2 -1070.215} C_VEL
LIN {X 0,Y 594.404,Z 533.089,A -85,B 0,C 180,E1 -1070.987,E2 -1070.987} C_VEL
LIN {X 0,Y 594.366,Z 541.984,A -85,B 0,C 180,E1 -1071.842,E2 -1071.842} C_VEL
LIN {X 0,Y 594.345,Z 550.67,A -85,B 0,C 180,E1 -1072.868,E2 -1072.868} C_VEL
LIN {X 0,Y 594.29,Z 557.599,A -85,B 0,C 180,E1 -1073.89,E2 -1073.89} C_VEL
LIN {X 0,Y 594.253,Z 563.151,A -85,B 0,C 180,E1 -1074.911,E2 -1074.911} C_VEL
LIN {X 0,Y 594.262,Z 567.513,A -85,B 0,C 180,E1 -1075.931,E2 -1075.931} C_VEL
LIN {X 0,Y 594.268,Z 569.816,A -85,B 0,C 180,E1 -1076.61,E2 -1076.61} C_VEL
LIN {X 0,Y 594.226,Z 571.694,A -85,B 0,C 180,E1 -1077.288,E2 -1077.288} C_VEL
LIN {X 0,Y 594.24,Z 573.127,A -85,B 0,C 180,E1 -1077.967,E2 -1077.967} C_VEL
LIN {X 0,Y 594.241,Z 574.753,A -85,B 0,C 180,E1 -1079.322,E2 -1079.322} C_VEL
LIN {X 0,Y 594.236,Z 574.996,A -85,B 0,C 180,E1 -1080,E2 -1080} C_VEL
LIN {X 0,Y 594.239,Z 574.815,A -85,B 0,C 180,E1 -1080.678,E2 -1080.678} C_VEL
LIN {X 0,Y 594.239,Z 573.275,A -85,B 0,C 180,E1 -1082.033,E2 -1082.033} C_VEL
LIN {X 0,Y 594.227,Z 571.915,A -85,B 0,C 180,E1 -1082.711,E2 -1082.711} C_VEL
LIN {X 0,Y 594.29,Z 569.038,A -85,B 0,C 180,E1 -1083.729,E2 -1083.729} C_VEL
LIN {X 0,Y 594.241,Z 565.139,A -85,B 0,C 180,E1 -1084.749,E2 -1084.749} C_VEL
LIN {X 0,Y 594.299,Z 560.107,A -85,B 0,C 180,E1 -1085.769,E2 -1085.769} C_VEL
LIN {X 0,Y 594.316,Z 553.788,A -85,B 0,C 180,E1 -1086.791,E2 -1086.791} C_VEL
LIN {X 0,Y 594.346,Z 545.87,A -85,B 0,C 180,E1 -1087.815,E2 -1087.815} C_VEL
LIN {X 0,Y 594.381,Z 536.024,A -85,B 0,C 180,E1 -1088.842,E2 -1088.842} C_VEL
LIN {X 0,Y 594.425,Z 525.703,A -85,B 0,C 180,E1 -1089.699,E2 -1089.699} C_VEL
LIN {X 0,Y 594.502,Z 514.08,A -85,B 0,C 180,E1 -1090.472,E2 -1090.472} C_VEL
LIN {X 0,Y 594.558,Z 502.066,A -85,B 0,C 180,E1 -1091.094,E2 -1091.094} C_VEL
LIN {X 0,Y 594.598,Z 489.232,A -85,B 0,C 180,E1 -1091.592,E2 -1091.592} C_VEL
LIN {X 0,Y 594.654,Z 476.6,A -85,B 0,C 180,E1 -1091.936,E2 -1091.936} C_VEL
LIN {X 0,Y 594.267,Z 471.673,A -85,B 0,C 180,E1 -1092.052,E2 -1092.052} C_VEL
LIN {X 0,Y 594.238,Z 468.458,A -85,B 0,C 180,E1 -1094.381,E2 -1094.381} C_VEL
LIN {X 0,Y 594.239,Z 464.613,A -85,B 0,C 180,E1 -1097.198,E2 -1097.198} C_VEL
LIN {X 0,Y 594.241,Z 461.729,A -85,B 0,C 180,E1 -1099.339,E2 -1099.339} C_VEL
LIN {X 0,Y 594.226,Z 458.845,A -85,B 0,C 180,E1 -1101.509,E2 -1101.509} C_VEL
LIN {X 0,Y 594.278,Z 455,A -85,B 0,C 180,E1 -1104.451,E2 -1104.451} C_VEL
LIN {X 0,Y 594.264,Z 452.115,A -85,B 0,C 180,E1 -1106.705,E2 -1106.705} C_VEL
LIN {X 0,Y 594.258,Z 449.25,A -85,B 0,C 180,E1 -1109.005,E2 -1109.005} C_VEL
LIN {X 0,Y 594.327,Z 446.789,A -85,B 0,C 180,E1 -1111.353,E2 -1111.353} C_VEL
LIN {X 0,Y 594.331,Z 443.668,A -85,B 0,C 180,E1 -1114.131,E2 -1114.131} C_VEL
LIN {X 0,Y 594.322,Z 442.458,A -85,B 0,C 180,E1 -1115.411,E2 -1115.411} C_VEL
LIN {X 0,Y 594.391,Z 442.449,A -85,B 0,C 180,E1 -1117.94,E2 -1117.94} C_VEL
LIN {X 0,Y 594.379,Z 442.448,A -85,B 0,C 180,E1 -1120.822,E2 -1120.822} C_VEL
LIN {X 0,Y 594.387,Z 442.45,A -85,B 0,C 180,E1 -1123.841,E2 -1123.841} C_VEL
LIN {X 0,Y 594.368,Z 442.449,A -85,B 0,C 180,E1 -1126.7,E2 -1126.7} C_VEL
LIN {X 0,Y 594.377,Z 442.448,A -85,B 0,C 180,E1 -1129.433,E2 -1129.433} C_VEL
LIN {X 0,Y 594.392,Z 442.449,A -85,B 0,C 180,E1 -1132.392,E2 -1132.392} C_VEL
LIN {X 0,Y 594.37,Z 442.557,A -85,B 0,C 180,E1 -1133.757,E2 -1133.757} C_VEL
LIN {X 0,Y 594.646,Z 444.949,A -85,B 0,C 180,E1 -1134.637,E2 -1134.637} C_VEL
LIN {X 0,Y 594.581,Z 452.394,A -85,B 0,C 180,E1 -1137.062,E2 -1137.062} C_VEL
LIN {X 0,Y 594.56,Z 462.148,A -85,B 0,C 180,E1 -1139.939,E2 -1139.939} C_VEL
LIN {X 0,Y 594.488,Z 472.422,A -85,B 0,C 180,E1 -1142.926,E2 -1142.926} C_VEL
LIN {X 0,Y 594.458,Z 481.69,A -85,B 0,C 180,E1 -1145.557,E2 -1145.557} C_VEL
LIN {X 0,Y 594.397,Z 492.281,A -85,B 0,C 180,E1 -1148.498,E2 -1148.498} C_VEL
LIN {X 0,Y 594.376,Z 502.872,A -85,B 0,C 180,E1 -1151.382,E2 -1151.382} C_VEL
LIN {X 0,Y 594.325,Z 513.463,A -85,B 0,C 180,E1 -1154.218,E2 -1154.218} C_VEL
LIN {X 0,Y 594.297,Z 524.054,A -85,B 0,C 180,E1 -1157.015,E2 -1157.015} C_VEL
LIN {X 0,Y 594.301,Z 527.53,A -85,B 0,C 180,E1 -1157.926,E2 -1157.926} C_VEL
LIN {X 0,Y 594.68,Z 533.223,A -85,B 0,C 180,E1 -1158.042,E2 -1158.042} C_VEL
LIN {X 0,Y 594.639,Z 546.492,A -85,B 0,C 180,E1 -1158.366,E2 -1158.366} C_VEL
LIN {X 0,Y 594.587,Z 558.361,A -85,B 0,C 180,E1 -1158.79,E2 -1158.79} C_VEL
LIN {X 0,Y 594.511,Z 570.207,A -85,B 0,C 180,E1 -1159.356,E2 -1159.356} C_VEL
LIN {X 0,Y 594.462,Z 581.475,A -85,B 0,C 180,E1 -1160.043,E2 -1160.043} C_VEL
LIN {X 0,Y 594.406,Z 591.645,A -85,B 0,C 180,E1 -1160.815,E2 -1160.815} C_VEL
LIN {X 0,Y 594.372,Z 600.786,A -85,B 0,C 180,E1 -1161.671,E2 -1161.671} C_VEL
LIN {X 0,Y 594.317,Z 609.69,A -85,B 0,C 180,E1 -1162.697,E2 -1162.697} C_VEL
LIN {X 0,Y 594.281,Z 616.168,A -85,B 0,C 180,E1 -1163.615,E2 -1163.615} C_VEL
LIN {X 0,Y 594.289,Z 621.68,A -85,B 0,C 180,E1 -1164.571,E2 -1164.571} C_VEL
LIN {X 0,Y 594.27,Z 626.371,A -85,B 0,C 180,E1 -1165.591,E2 -1165.591} C_VEL
LIN {X 0,Y 594.267,Z 629.956,A -85,B 0,C 180,E1 -1166.61,E2 -1166.61} C_VEL
LIN {X 0,Y 594.226,Z 631.809,A -85,B 0,C 180,E1 -1167.288,E2 -1167.288} C_VEL
LIN {X 0,Y 594.24,Z 633.201,A -85,B 0,C 180,E1 -1167.967,E2 -1167.967} C_VEL
LIN {X 0,Y 594.239,Z 634.784,A -85,B 0,C 180,E1 -1169.322,E2 -1169.322} C_VEL
LIN {X 0,Y 594.236,Z 635,A -85,B 0,C 180,E1 -1170,E2 -1170} C_VEL
LIN {X 0,Y 594.247,Z 634.185,A -85,B 0,C 180,E1 -1171.355,E2 -1171.355} C_VEL
LIN {X 0,Y 594.24,Z 633.202,A -85,B 0,C 180,E1 -1172.033,E2 -1172.033} C_VEL
LIN {X 0,Y 594.226,Z 631.81,A -85,B 0,C 180,E1 -1172.712,E2 -1172.712} C_VEL
LIN {X 0,Y 594.288,Z 628.896,A -85,B 0,C 180,E1 -1173.729,E2 -1173.729} C_VEL
LIN {X 0,Y 594.242,Z 624.95,A -85,B 0,C 180,E1 -1174.749,E2 -1174.749} C_VEL
LIN {X 0,Y 594.304,Z 618.878,A -85,B 0,C 180,E1 -1175.939,E2 -1175.939} C_VEL
LIN {X 0,Y 594.308,Z 612.236,A -85,B 0,C 180,E1 -1176.962,E2 -1176.962} C_VEL
LIN {X 0,Y 594.359,Z 603.99,A -85,B 0,C 180,E1 -1177.986,E2 -1177.986} C_VEL
LIN {X 0,Y 594.382,Z 595.537,A -85,B 0,C 180,E1 -1178.842,E2 -1178.842} C_VEL
LIN {X 0,Y 594.431,Z 585.094,A -85,B 0,C 180,E1 -1179.699,E2 -1179.699} C_VEL
LIN {X 0,Y 594.482,Z 574.759,A -85,B 0,C 180,E1 -1180.386,E2 -1180.386} C_VEL
LIN {X 0,Y 594.534,Z 563.748,A -85,B 0,C 180,E1 -1180.972,E2 -1180.972} C_VEL
LIN {X 0,Y 594.598,Z 551.719,A -85,B 0,C 180,E1 -1181.464,E2 -1181.464} C_VEL
LIN {X 0,Y 594.655,Z 538.353,A -85,B 0,C 180,E1 -1181.85,E2 -1181.85} C_VEL
LIN {X 0,Y 594.455,Z 528.769,A -85,B 0,C 180,E1 -1182.039,E2 -1182.039} C_VEL
LIN {X 0,Y 594.301,Z 527.53,A -85,B 0,C 180,E1 -1182.073,E2 -1182.073} C_VEL
LIN {X 0,Y 594.317,Z 517.436,A -85,B 0,C 180,E1 -1184.729,E2 -1184.729} C_VEL
LIN {X 0,Y 594.334,Z 506.844,A -85,B 0,C 180,E1 -1187.55,E2 -1187.55} C_VEL
LIN {X 0,Y 594.381,Z 496.253,A -85,B 0,C 180,E1 -1190.415,E2 -1190.415} C_VEL
LIN {X 0,Y 594.437,Z 485.662,A -85,B 0,C 180,E1 -1193.333,E2 -1193.333} C_VEL
LIN {X 0,Y 594.484,Z 476.035,A -85,B 0,C 180,E1 -1196.041,E2 -1196.041} C_VEL
LIN {X 0,Y 594.507,Z 467.144,A -85,B 0,C 180,E1 -1198.601,E2 -1198.601} C_VEL
LIN {X 0,Y 594.577,Z 457.787,A -85,B 0,C 180,E1 -1201.338,E2 -1201.338} C_VEL
LIN {X 0,Y 594.66,Z 448.494,A -85,B 0,C 180,E1 -1204.178,E2 -1204.178} C_VEL
LIN {X 0,Y 594.431,Z 442.695,A -85,B 0,C 180,E1 -1206.029,E2 -1206.029} C_VEL
LIN {X 0,Y 594.356,Z 442.452,A -85,B 0,C 180,E1 -1206.244,E2 -1206.244} C_VEL
LIN {X 0,Y 594.388,Z 442.445,A -85,B 0,C 180,E1 -1208.805,E2 -1208.805} C_VEL
LIN {X 0,Y 594.383,Z 442.446,A -85,B 0,C 180,E1 -1211.848,E2 -1211.848} C_VEL
LIN {X 0,Y 594.366,Z 442.449,A -85,B 0,C 180,E1 -1214.809,E2 -1214.809} C_VEL
LIN {X 0,Y 594.374,Z 442.452,A -85,B 0,C 180,E1 -1217.625,E2 -1217.625} C_VEL
LIN {X 0,Y 594.372,Z 442.447,A -85,B 0,C 180,E1 -1220.319,E2 -1220.319} C_VEL
LIN {X 0,Y 594.385,Z 442.444,A -85,B 0,C 180,E1 -1222.913,E2 -1222.913} C_VEL
LIN {X 0,Y 594.385,Z 442.446,A -85,B 0,C 180,E1 -1225.861,E2 -1225.861} C_VEL
LIN {X 0,Y 594.371,Z 442.451,A -85,B 0,C 180,E1 -1228.65,E2 -1228.65} C_VEL
LIN {X 0,Y 594.386,Z 442.444,A -85,B 0,C 180,E1 -1231.042,E2 -1231.042} C_VEL
LIN {X 0,Y 594.386,Z 442.444,A -85,B 0,C 180,E1 -1233.978,E2 -1233.978} C_VEL
LIN {X 0,Y 594.389,Z 442.449,A -85,B 0,C 180,E1 -1236.296,E2 -1236.296} C_VEL
LIN {X 0,Y 594.407,Z 442.444,A -85,B 0,C 180,E1 -1239.225,E2 -1239.225} C_VEL
LIN {X 0,Y 594.353,Z 442.449,A -85,B 0,C 180,E1 -1242.095,E2 -1242.095} C_VEL
LIN {X 0,Y 594.369,Z 442.452,A -85,B 0,C 180,E1 -1244.219,E2 -1244.219} C_VEL
LIN {X 0,Y 594.371,Z 442.449,A -85,B 0,C 180,E1 -1247.017,E2 -1247.017} C_VEL
LIN {X 0,Y 594.392,Z 442.443,A -85,B 0,C 180,E1 -1249.784,E2 -1249.784} C_VEL
LIN {X 0,Y 594.396,Z 442.443,A -85,B 0,C 180,E1 -1252.527,E2 -1252.527} C_VEL
LIN {X 0,Y 594.398,Z 442.447,A -85,B 0,C 180,E1 -1255.253,E2 -1255.253} C_VEL
LIN {X 0,Y 594.394,Z 442.446,A -85,B 0,C 180,E1 -1257.967,E2 -1257.967} C_VEL
LIN {X 0,Y 594.425,Z 442.439,A -85,B 0,C 180,E1 -1260.678,E2 -1260.678} C_VEL
LIN {X 0,Y 594.38,Z 442.445,A -85,B 0,C 180,E1 -1263.389,E2 -1263.389} C_VEL
LIN {X 0,Y 594.37,Z 442.451,A -85,B 0,C 180,E1 -1266.109,E2 -1266.109} C_VEL
LIN {X 0,Y 594.4,Z 442.445,A -85,B 0,C 180,E1 -1268.842,E2 -1268.842} C_VEL
LIN {X 0,Y 594.388,Z 442.443,A -85,B 0,C 180,E1 -1271.596,E2 -1271.596} C_VEL
LIN {X 0,Y 594.393,Z 442.444,A -85,B 0,C 180,E1 -1274.377,E2 -1274.377} C_VEL
LIN {X 0,Y 594.362,Z 442.448,A -85,B 0,C 180,E1 -1275.327,E2 -1275.327} C_VEL
LIN {X 0,Y 593.686,Z 442.533,A -85,B 0,C 180,E1 -1275.893,E2 -1275.893} C_VEL
LIN {X 0,Y 590.82,Z 442.893,A -85,B 0,C 180,E1 -1276.811,E2 -1276.811} C_VEL
LIN {X 0,Y 588.41,Z 443.192,A -85,B 0,C 180,E1 -1277.55,E2 -1277.55} C_VEL
LIN {X 0,Y 587.388,Z 443.317,A -85,B 0,C 180,E1 -1278.12,E2 -1278.12} C_VEL
LIN {X 0,Y 587.311,Z 443.326,A -85,B 0,C 180,E1 -1278.313,E2 -1278.313} C_VEL
LIN {X 0,Y 587.334,Z 443.323,A -85,B 0,C 180,E1 -1281.038,E2 -1281.038} C_VEL
LIN {X 0,Y 587.324,Z 443.329,A -85,B 0,C 180,E1 -1283.259,E2 -1283.259} C_VEL
LIN {X 0,Y 587.335,Z 443.322,A -85,B 0,C 180,E1 -1285.517,E2 -1285.517} C_VEL
LIN {X 0,Y 587.352,Z 443.326,A -85,B 0,C 180,E1 -1287.818,E2 -1287.818} C_VEL
LIN {X 0,Y 587.34,Z 443.323,A -85,B 0,C 180,E1 -1290.51,E2 -1290.51} C_VEL
LIN {X 0,Y 587.339,Z 443.321,A -85,B 0,C 180,E1 -1293.397,E2 -1293.397} C_VEL
LIN {X 0,Y 587.351,Z 443.324,A -85,B 0,C 180,E1 -1295.896,E2 -1295.896} C_VEL
LIN {X 0,Y 587.331,Z 443.325,A -85,B 0,C 180,E1 -1298.48,E2 -1298.48} C_VEL
LIN {X 0,Y 587.339,Z 443.322,A -85,B 0,C 180,E1 -1301.157,E2 -1301.157} C_VEL
LIN {X 0,Y 587.339,Z 443.322,A -85,B 0,C 180,E1 -1304.114,E2 -1304.114} C_VEL
LIN {X 0,Y 587.315,Z 443.326,A -85,B 0,C 180,E1 -1306.994,E2 -1306.994} C_VEL
LIN {X 0,Y 587.317,Z 443.33,A -85,B 0,C 180,E1 -1309.746,E2 -1309.746} C_VEL
LIN {X 0,Y 587.349,Z 443.322,A -85,B 0,C 180,E1 -1312.393,E2 -1312.393} C_VEL
LIN {X 0,Y 587.36,Z 443.322,A -85,B 0,C 180,E1 -1315.651,E2 -1315.651} C_VEL
LIN {X 0,Y 587.347,Z 443.321,A -85,B 0,C 180,E1 -1318.231,E2 -1318.231} C_VEL
LIN {X 0,Y 587.355,Z 443.323,A -85,B 0,C 180,E1 -1320.867,E2 -1320.867} C_VEL
LIN {X 0,Y 587.363,Z 443.324,A -85,B 0,C 180,E1 -1323.819,E2 -1323.819} C_VEL
LIN {X 0,Y 587.34,Z 443.322,A -85,B 0,C 180,E1 -1325.994,E2 -1325.994} C_VEL
LIN {X 0,Y 587.321,Z 443.328,A -85,B 0,C 180,E1 -1328.226,E2 -1328.226} C_VEL
LIN {X 0,Y 587.353,Z 443.322,A -85,B 0,C 180,E1 -1331.151,E2 -1331.151} C_VEL
LIN {X 0,Y 587.323,Z 443.324,A -85,B 0,C 180,E1 -1334.025,E2 -1334.025} C_VEL
LIN {X 0,Y 587.364,Z 443.324,A -85,B 0,C 180,E1 -1336.154,E2 -1336.154} C_VEL
LIN {X 0,Y 587.347,Z 443.323,A -85,B 0,C 180,E1 -1338.963,E2 -1338.963} C_VEL
LIN {X 0,Y 587.37,Z 443.318,A -85,B 0,C 180,E1 -1341.745,E2 -1341.745} C_VEL
LIN {X 0,Y 587.358,Z 443.32,A -85,B 0,C 180,E1 -1344.507,E2 -1344.507} C_VEL
LIN {X 0,Y 587.374,Z 443.322,A -85,B 0,C 180,E1 -1347.257,E2 -1347.257} C_VEL
LIN {X 0,Y 587.389,Z 443.319,A -85,B 0,C 180,E1 -1350,E2 -1350} C_VEL
LIN {X 0,Y 587.372,Z 443.318,A -85,B 0,C 180,E1 -1352.743,E2 -1352.743} C_VEL
LIN {X 0,Y 587.359,Z 443.32,A -85,B 0,C 180,E1 -1355.493,E2 -1355.493} C_VEL
LIN {X 0,Y 587.347,Z 443.324,A -85,B 0,C 180,E1 -1358.256,E2 -1358.256} C_VEL
LIN {X 0,Y 587.355,Z 443.326,A -85,B 0,C 180,E1 -1361.134,E2 -1361.134} C_VEL
LIN {X 0,Y 587.371,Z 443.324,A -85,B 0,C 180,E1 -1364.26,E2 -1364.26} C_VEL
LIN {X 0,Y 587.349,Z 443.327,A -85,B 0,C 180,E1 -1367.406,E2 -1367.406} C_VEL
LIN {X 0,Y 587.335,Z 443.326,A -85,B 0,C 180,E1 -1370.305,E2 -1370.305} C_VEL
LIN {X 0,Y 587.327,Z 443.325,A -85,B 0,C 180,E1 -1373.259,E2 -1373.259} C_VEL
LIN {X 0,Y 587.339,Z 443.324,A -85,B 0,C 180,E1 -1375.517,E2 -1375.517} C_VEL
LIN {X 0,Y 587.346,Z 443.322,A -85,B 0,C 180,E1 -1377.818,E2 -1377.818} C_VEL
LIN {X 0,Y 587.341,Z 443.321,A -85,B 0,C 180,E1 -1380.51,E2 -1380.51} C_VEL
LIN {X 0,Y 587.338,Z 443.324,A -85,B 0,C 180,E1 -1383.397,E2 -1383.397} C_VEL
LIN {X 0,Y 587.297,Z 443.33,A -85,B 0,C 180,E1 -1385.9,E2 -1385.9} C_VEL
LIN {X 0,Y 587.33,Z 443.323,A -85,B 0,C 180,E1 -1388.48,E2 -1388.48} C_VEL
LIN {X 0,Y 587.339,Z 443.324,A -85,B 0,C 180,E1 -1391.157,E2 -1391.157} C_VEL
LIN {X 0,Y 587.316,Z 443.328,A -85,B 0,C 180,E1 -1394.112,E2 -1394.112} C_VEL
LIN {X 0,Y 587.322,Z 443.33,A -85,B 0,C 180,E1 -1396.994,E2 -1396.994} C_VEL
LIN {X 0,Y 587.316,Z 443.326,A -85,B 0,C 180,E1 -1399.745,E2 -1399.745} C_VEL
LIN {X 0,Y 587.348,Z 443.32,A -85,B 0,C 180,E1 -1402.392,E2 -1402.392} C_VEL
LIN {X 0,Y 587.257,Z 443.338,A -85,B 0,C 180,E1 -1404.939,E2 -1404.939} C_VEL
LIN {X 0,Y 587.266,Z 443.567,A -85,B 0,C 180,E1 -1405.773,E2 -1405.773} C_VEL
LIN {X 0,Y 587.22,Z 446.421,A -85,B 0,C 180,E1 -1408.223,E2 -1408.223} C_VEL
LIN {X 0,Y 587.179,Z 449.624,A -85,B 0,C 180,E1 -1410.897,E2 -1410.897} C_VEL
LIN {X 0,Y 587.164,Z 452.002,A -85,B 0,C 180,E1 -1412.945,E2 -1412.945} C_VEL
LIN {X 0,Y 587.196,Z 455.164,A -85,B 0,C 180,E1 -1415.454,E2 -1415.454} C_VEL
LIN {X 0,Y 587.142,Z 458.727,A -85,B 0,C 180,E1 -1418.218,E2 -1418.218} C_VEL
LIN {X 0,Y 587.153,Z 462.399,A -85,B 0,C 180,E1 -1421.015,E2 -1421.015} C_VEL
LIN {X 0,Y 587.155,Z 466.414,A -85,B 0,C 180,E1 -1424.02,E2 -1424.02} C_VEL
LIN {X 0,Y 587.14,Z 470.257,A -85,B 0,C 180,E1 -1426.854,E2 -1426.854} C_VEL
LIN {X 0,Y 587.156,Z 471.668,A -85,B 0,C 180,E1 -1427.887,E2 -1427.887} C_VEL
LIN {X 0,Y 587.701,Z 477.377,A -85,B 0,C 180,E1 -1428.03,E2 -1428.03} C_VEL
LIN {X 0,Y 587.65,Z 490.665,A -85,B 0,C 180,E1 -1428.408,E2 -1428.408} C_VEL
LIN {X 0,Y 587.574,Z 502.908,A -85,B 0,C 180,E1 -1428.901,E2 -1428.901} C_VEL
LIN {X 0,Y 587.483,Z 515.439,A -85,B 0,C 180,E1 -1429.575,E2 -1429.575} C_VEL
LIN {X 0,Y 587.393,Z 526.813,A -85,B 0,C 180,E1 -1430.357,E2 -1430.357} C_VEL
LIN {X 0,Y 587.337,Z 536.874,A -85,B 0,C 180,E1 -1431.224,E2 -1431.224} C_VEL
LIN {X 0,Y 587.274,Z 546.576,A -85,B 0,C 180,E1 -1432.263,E2 -1432.263} C_VEL
LIN {X 0,Y 587.236,Z 553.148,A -85,B 0,C 180,E1 -1433.126,E2 -1433.126} C_VEL
LIN {X 0,Y 587.237,Z 559.617,A -85,B 0,C 180,E1 -1434.161,E2 -1434.161} C_VEL
LIN {X 0,Y 587.146,Z 564.757,A -85,B 0,C 180,E1 -1435.194,E2 -1435.194} C_VEL
LIN {X 0,Y 587.213,Z 568.747,A -85,B 0,C 180,E1 -1436.226,E2 -1436.226} C_VEL
LIN {X 0,Y 587.132,Z 571.696,A -85,B 0,C 180,E1 -1437.255,E2 -1437.255} C_VEL
LIN {X 0,Y 587.139,Z 573.127,A -85,B 0,C 180,E1 -1437.942,E2 -1437.942} C_VEL
LIN {X 0,Y 587.141,Z 574.754,A -85,B 0,C 180,E1 -1439.314,E2 -1439.314} C_VEL
LIN {X 0,Y 587.137,Z 574.996,A -85,B 0,C 180,E1 -1440,E2 -1440} C_VEL
LIN {X 0,Y 587.14,Z 574.815,A -85,B 0,C 180,E1 -1440.686,E2 -1440.686} C_VEL
LIN {X 0,Y 587.138,Z 573.274,A -85,B 0,C 180,E1 -1442.058,E2 -1442.058} C_VEL
LIN {X 0,Y 587.133,Z 571.913,A -85,B 0,C 180,E1 -1442.744,E2 -1442.744} C_VEL
LIN {X 0,Y 587.213,Z 569.036,A -85,B 0,C 180,E1 -1443.774,E2 -1443.774} C_VEL
LIN {X 0,Y 587.147,Z 565.136,A -85,B 0,C 180,E1 -1444.806,E2 -1444.806} C_VEL
LIN {X 0,Y 587.23,Z 560.105,A -85,B 0,C 180,E1 -1445.839,E2 -1445.839} C_VEL
LIN {X 0,Y 587.23,Z 553.784,A -85,B 0,C 180,E1 -1446.874,E2 -1446.874} C_VEL
LIN {X 0,Y 587.288,Z 545.866,A -85,B 0,C 180,E1 -1447.91,E2 -1447.91} C_VEL
LIN {X 0,Y 587.343,Z 536.018,A -85,B 0,C 180,E1 -1448.949,E2 -1448.949} C_VEL
LIN {X 0,Y 587.409,Z 525.697,A -85,B 0,C 180,E1 -1449.816,E2 -1449.816} C_VEL
LIN {X 0,Y 587.505,Z 514.069,A -85,B 0,C 180,E1 -1450.598,E2 -1450.598} C_VEL
LIN {X 0,Y 587.586,Z 502.43,A -85,B 0,C 180,E1 -1451.211,E2 -1451.211} C_VEL
LIN {X 0,Y 587.622,Z 490.587,A -85,B 0,C 180,E1 -1451.685,E2 -1451.685} C_VEL
LIN {X 0,Y 587.712,Z 477.492,A -85,B 0,C 180,E1 -1452.058,E2 -1452.058} C_VEL
LIN {X 0,Y 587.289,Z 472.863,A -85,B 0,C 180,E1 -1452.162,E2 -1452.162} C_VEL
LIN {X 0,Y 587.158,Z 471.642,A -85,B 0,C 180,E1 -1452.223,E2 -1452.223} C_VEL
LIN {X 0,Y 587.131,Z 468.458,A -85,B 0,C 180,E1 -1454.559,E2 -1454.559} C_VEL
LIN {X 0,Y 587.147,Z 465.503,A -85,B 0,C 180,E1 -1456.747,E2 -1456.747} C_VEL
LIN {X 0,Y 587.135,Z 461.728,A -85,B 0,C 180,E1 -1459.582,E2 -1459.582} C_VEL
LIN {X 0,Y 587.143,Z 458.844,A -85,B 0,C 180,E1 -1461.781,E2 -1461.781} C_VEL
LIN {X 0,Y 587.179,Z 454.999,A -85,B 0,C 180,E1 -1464.766,E2 -1464.766} C_VEL
LIN {X 0,Y 587.166,Z 452.114,A -85,B 0,C 180,E1 -1467.054,E2 -1467.054} C_VEL
LIN {X 0,Y 587.2,Z 449.667,A -85,B 0,C 180,E1 -1469.388,E2 -1469.388} C_VEL
LIN {X 0,Y 587.269,Z 446.953,A -85,B 0,C 180,E1 -1471.823,E2 -1471.823} C_VEL
LIN {X 0,Y 587.272,Z 444.185,A -85,B 0,C 180,E1 -1474.336,E2 -1474.336} C_VEL
LIN {X 0,Y 587.238,Z 443.377,A -85,B 0,C 180,E1 -1475.062,E2 -1475.062} C_VEL
LIN {X 0,Y 587.349,Z 443.325,A -85,B 0,C 180,E1 -1477.607,E2 -1477.607} C_VEL
LIN {X 0,Y 587.315,Z 443.331,A -85,B 0,C 180,E1 -1480.254,E2 -1480.254} C_VEL
LIN {X 0,Y 587.326,Z 443.327,A -85,B 0,C 180,E1 -1483.006,E2 -1483.006} C_VEL
LIN {X 0,Y 587.33,Z 443.326,A -85,B 0,C 180,E1 -1485.887,E2 -1485.887} C_VEL
LIN {X 0,Y 587.341,Z 443.326,A -85,B 0,C 180,E1 -1488.925,E2 -1488.925} C_VEL
LIN {X 0,Y 587.335,Z 443.327,A -85,B 0,C 180,E1 -1491.521,E2 -1491.521} C_VEL
LIN {X 0,Y 587.362,Z 443.398,A -85,B 0,C 180,E1 -1493.467,E2 -1493.467} C_VEL
LIN {X 0,Y 587.704,Z 445.818,A -85,B 0,C 180,E1 -1494.407,E2 -1494.407} C_VEL
LIN {X 0,Y 587.611,Z 453.051,A -85,B 0,C 180,E1 -1496.848,E2 -1496.848} C_VEL
LIN {X 0,Y 587.582,Z 463.048,A -85,B 0,C 180,E1 -1499.844,E2 -1499.844} C_VEL
LIN {X 0,Y 587.5,Z 473.746,A -85,B 0,C 180,E1 -1502.962,E2 -1502.962} C_VEL
LIN {X 0,Y 587.428,Z 483.289,A -85,B 0,C 180,E1 -1505.7,E2 -1505.7} C_VEL
LIN {X 0,Y 587.358,Z 493.606,A -85,B 0,C 180,E1 -1508.596,E2 -1508.596} C_VEL
LIN {X 0,Y 587.323,Z 504.196,A -85,B 0,C 180,E1 -1511.512,E2 -1511.512} C_VEL
LIN {X 0,Y 587.261,Z 514.787,A -85,B 0,C 180,E1 -1514.379,E2 -1514.379} C_VEL
LIN {X 0,Y 587.24,Z 524.054,A -85,B 0,C 180,E1 -1516.856,E2 -1516.856} C_VEL
LIN {X 0,Y 587.215,Z 527.571,A -85,B 0,C 180,E1 -1517.789,E2 -1517.789} C_VEL
LIN {X 0,Y 587.736,Z 533.223,A -85,B 0,C 180,E1 -1517.899,E2 -1517.899} C_VEL
LIN {X 0,Y 587.684,Z 546.493,A -85,B 0,C 180,E1 -1518.226,E2 -1518.226} C_VEL
LIN {X 0,Y 587.623,Z 558.272,A -85,B 0,C 180,E1 -1518.651,E2 -1518.651} C_VEL
LIN {X 0,Y 587.528,Z 570.208,A -85,B 0,C 180,E1 -1519.228,E2 -1519.228} C_VEL
LIN {X 0,Y 587.457,Z 581.476,A -85,B 0,C 180,E1 -1519.923,E2 -1519.923} C_VEL
LIN {X 0,Y 587.384,Z 591.646,A -85,B 0,C 180,E1 -1520.704,E2 -1520.704} C_VEL
LIN {X 0,Y 587.34,Z 600.786,A -85,B 0,C 180,E1 -1521.571,E2 -1521.571} C_VEL
LIN {X 0,Y 587.259,Z 609.69,A -85,B 0,C 180,E1 -1522.608,E2 -1522.608} C_VEL
LIN {X 0,Y 587.195,Z 616.745,A -85,B 0,C 180,E1 -1523.627,E2 -1523.627} C_VEL
LIN {X 0,Y 587.211,Z 621.68,A -85,B 0,C 180,E1 -1524.506,E2 -1524.506} C_VEL
LIN {X 0,Y 587.188,Z 626.371,A -85,B 0,C 180,E1 -1525.538,E2 -1525.538} C_VEL
LIN {X 0,Y 587.194,Z 629.956,A -85,B 0,C 180,E1 -1526.569,E2 -1526.569} C_VEL
LIN {X 0,Y 587.132,Z 631.808,A -85,B 0,C 180,E1 -1527.256,E2 -1527.256} C_VEL
LIN {X 0,Y 587.139,Z 633.201,A -85,B 0,C 180,E1 -1527.942,E2 -1527.942} C_VEL
LIN {X 0,Y 587.14,Z 634.784,A -85,B 0,C 180,E1 -1529.314,E2 -1529.314} C_VEL
LIN {X 0,Y 587.137,Z 635,A -85,B 0,C 180,E1 -1530,E2 -1530} C_VEL
LIN {X 0,Y 587.147,Z 634.185,A -85,B 0,C 180,E1 -1531.372,E2 -1531.372} C_VEL
LIN {X 0,Y 587.139,Z 633.201,A -85,B 0,C 180,E1 -1532.058,E2 -1532.058} C_VEL
LIN {X 0,Y 587.132,Z 631.81,A -85,B 0,C 180,E1 -1532.744,E2 -1532.744} C_VEL
LIN {X 0,Y 587.212,Z 628.896,A -85,B 0,C 180,E1 -1533.774,E2 -1533.774} C_VEL
LIN {X 0,Y 587.147,Z 624.95,A -85,B 0,C 180,E1 -1534.806,E2 -1534.806} C_VEL
LIN {X 0,Y 587.217,Z 618.878,A -85,B 0,C 180,E1 -1536.011,E2 -1536.011} C_VEL
LIN {X 0,Y 587.245,Z 612.237,A -85,B 0,C 180,E1 -1537.046,E2 -1537.046} C_VEL
LIN {X 0,Y 587.299,Z 603.99,A -85,B 0,C 180,E1 -1538.083,E2 -1538.083} C_VEL
LIN {X 0,Y 587.343,Z 595.538,A -85,B 0,C 180,E1 -1538.949,E2 -1538.949} C_VEL
LIN {X 0,Y 587.417,Z 585.095,A -85,B 0,C 180,E1 -1539.816,E2 -1539.816} C_VEL
LIN {X 0,Y 587.501,Z 574.759,A -85,B 0,C 180,E1 -1540.511,E2 -1540.511} C_VEL
LIN {X 0,Y 587.557,Z 562.855,A -85,B 0,C 180,E1 -1541.147,E2 -1541.147} C_VEL
LIN {X 0,Y 587.637,Z 550.62,A -85,B 0,C 180,E1 -1541.638,E2 -1541.638} C_VEL
LIN {X 0,Y 587.722,Z 537.438,A -85,B 0,C 180,E1 -1542.014,E2 -1542.014} C_VEL
LIN {X 0,Y 587.517,Z 529.615,A -85,B 0,C 180,E1 -1542.171,E2 -1542.171} C_VEL
LIN {X 0,Y 587.214,Z 527.53,A -85,B 0,C 180,E1 -1542.221,E2 -1542.221} C_VEL
LIN {X 0,Y 587.269,Z 517.436,A -85,B 0,C 180,E1 -1544.91,E2 -1544.91} C_VEL
LIN {X 0,Y 587.302,Z 506.844,A -85,B 0,C 180,E1 -1547.767,E2 -1547.767} C_VEL
LIN {X 0,Y 587.375,Z 496.253,A -85,B 0,C 180,E1 -1550.669,E2 -1550.669} C_VEL
LIN {X 0,Y 587.432,Z 485.662,A -85,B 0,C 180,E1 -1553.628,E2 -1553.628} C_VEL
LIN {X 0,Y 587.485,Z 476.395,A -85,B 0,C 180,E1 -1556.272,E2 -1556.272} C_VEL
LIN {X 0,Y 587.51,Z 468.451,A -85,B 0,C 180,E1 -1558.587,E2 -1558.587} C_VEL
LIN {X 0,Y 587.605,Z 459.051,A -85,B 0,C 180,E1 -1561.351,E2 -1561.351} C_VEL
LIN {X 0,Y 587.722,Z 449.88,A -85,B 0,C 180,E1 -1564.196,E2 -1564.196} C_VEL
LIN {X 0,Y 587.577,Z 444.666,A -85,B 0,C 180,E1 -1565.88,E2 -1565.88} C_VEL
LIN {X 0,Y 587.334,Z 443.328,A -85,B 0,C 180,E1 -1566.37,E2 -1566.37} C_VEL
LIN {X 0,Y 587.335,Z 443.323,A -85,B 0,C 180,E1 -1568.942,E2 -1568.942} C_VEL
LIN {X 0,Y 587.339,Z 443.325,A -85,B 0,C 180,E1 -1571.157,E2 -1571.157} C_VEL
LIN {X 0,Y 587.328,Z 443.324,A -85,B 0,C 180,E1 -1574.113,E2 -1574.113} C_VEL
LIN {X 0,Y 587.325,Z 443.324,A -85,B 0,C 180,E1 -1576.994,E2 -1576.994} C_VEL
LIN {X 0,Y 587.314,Z 443.325,A -85,B 0,C 180,E1 -1579.746,E2 -1579.746} C_VEL
LIN {X 0,Y 587.346,Z 443.327,A -85,B 0,C 180,E1 -1582.392,E2 -1582.392} C_VEL
LIN {X 0,Y 587.351,Z 443.324,A -85,B 0,C 180,E1 -1585.652,E2 -1585.652} C_VEL
LIN {X 0,Y 587.344,Z 443.323,A -85,B 0,C 180,E1 -1588.231,E2 -1588.231} C_VEL
LIN {X 0,Y 587.353,Z 443.32,A -85,B 0,C 180,E1 -1590.866,E2 -1590.866} C_VEL
LIN {X 0,Y 587.361,Z 443.319,A -85,B 0,C 180,E1 -1593.819,E2 -1593.819} C_VEL
LIN {X 0,Y 587.337,Z 443.323,A -85,B 0,C 180,E1 -1595.994,E2 -1595.994} C_VEL
LIN {X 0,Y 587.328,Z 443.326,A -85,B 0,C 180,E1 -1598.226,E2 -1598.226} C_VEL
LIN {X 0,Y 587.352,Z 443.325,A -85,B 0,C 180,E1 -1601.151,E2 -1601.151} C_VEL
LIN {X 0,Y 587.327,Z 443.327,A -85,B 0,C 180,E1 -1604.025,E2 -1604.025} C_VEL
LIN {X 0,Y 587.363,Z 443.32,A -85,B 0,C 180,E1 -1606.154,E2 -1606.154} C_VEL
LIN {X 0,Y 587.345,Z 443.326,A -85,B 0,C 180,E1 -1608.963,E2 -1608.963} C_VEL
LIN {X 0,Y 587.369,Z 443.321,A -85,B 0,C 180,E1 -1611.745,E2 -1611.745} C_VEL
LIN {X 0,Y 587.36,Z 443.32,A -85,B 0,C 180,E1 -1614.507,E2 -1614.507} C_VEL
LIN {X 0,Y 587.377,Z 443.317,A -85,B 0,C 180,E1 -1617.257,E2 -1617.257} C_VEL
LIN {X 0,Y 587.386,Z 443.319,A -85,B 0,C 180,E1 -1620,E2 -1620} C_VEL
LIN {X 0,Y 587.381,Z 443.321,A -85,B 0,C 180,E1 -1622.743,E2 -1622.743} C_VEL
LIN {X 0,Y 587.357,Z 443.32,A -85,B 0,C 180,E1 -1625.493,E2 -1625.493} C_VEL
LIN {X 0,Y 587.372,Z 443.318,A -85,B 0,C 180,E1 -1628.255,E2 -1628.255} C_VEL
LIN {X 0,Y 587.352,Z 443.321,A -85,B 0,C 180,E1 -1631.134,E2 -1631.134} C_VEL
LIN {X 0,Y 587.369,Z 443.319,A -85,B 0,C 180,E1 -1634.261,E2 -1634.261} C_VEL
LIN {X 0,Y 587.352,Z 443.321,A -85,B 0,C 180,E1 -1637.406,E2 -1637.406} C_VEL
LIN {X 0,Y 587.311,Z 443.326,A -85,B 0,C 180,E1 -1638.313,E2 -1638.313} C_VEL
LIN {X 0,Y 586.669,Z 443.407,A -85,B 0,C 180,E1 -1638.885,E2 -1638.885} C_VEL
LIN {X 0,Y 583.845,Z 443.761,A -85,B 0,C 180,E1 -1639.814,E2 -1639.814} C_VEL
LIN {X 0,Y 581.434,Z 444.063,A -85,B 0,C 180,E1 -1640.561,E2 -1640.561} C_VEL
LIN {X 0,Y 580.381,Z 444.192,A -85,B 0,C 180,E1 -1641.137,E2 -1641.137} C_VEL
LIN {X 0,Y 580.287,Z 444.203,A -85,B 0,C 180,E1 -1641.333,E2 -1641.333} C_VEL
LIN {X 0,Y 580.303,Z 444.2,A -85,B 0,C 180,E1 -1644.316,E2 -1644.316} C_VEL
LIN {X 0,Y 580.279,Z 444.203,A -85,B 0,C 180,E1 -1646.624,E2 -1646.624} C_VEL
LIN {X 0,Y 580.305,Z 444.203,A -85,B 0,C 180,E1 -1649.31,E2 -1649.31} C_VEL
LIN {X 0,Y 580.303,Z 444.2,A -85,B 0,C 180,E1 -1652.201,E2 -1652.201} C_VEL
LIN {X 0,Y 580.293,Z 444.2,A -85,B 0,C 180,E1 -1654.696,E2 -1654.696} C_VEL
LIN {X 0,Y 580.304,Z 444.204,A -85,B 0,C 180,E1 -1657.268,E2 -1657.268} C_VEL
LIN {X 0,Y 580.293,Z 444.205,A -85,B 0,C 180,E1 -1660.27,E2 -1660.27} C_VEL
LIN {X 0,Y 580.285,Z 444.201,A -85,B 0,C 180,E1 -1662.706,E2 -1662.706} C_VEL
LIN {X 0,Y 580.274,Z 444.202,A -85,B 0,C 180,E1 -1665.609,E2 -1665.609} C_VEL
LIN {X 0,Y 580.283,Z 444.206,A -85,B 0,C 180,E1 -1668.231,E2 -1668.231} C_VEL
LIN {X 0,Y 580.282,Z 444.204,A -85,B 0,C 180,E1 -1670.965,E2 -1670.965} C_VEL
LIN {X 0,Y 580.273,Z 444.202,A -85,B 0,C 180,E1 -1673.597,E2 -1673.597} C_VEL
LIN {X 0,Y 580.323,Z 444.199,A -85,B 0,C 180,E1 -1676.146,E2 -1676.146} C_VEL
LIN {X 0,Y 580.28,Z 444.203,A -85,B 0,C 180,E1 -1678.615,E2 -1678.615} C_VEL
LIN {X 0,Y 580.297,Z 444.2,A -85,B 0,C 180,E1 -1681.024,E2 -1681.024} C_VEL
LIN {X 0,Y 580.295,Z 444.204,A -85,B 0,C 180,E1 -1683.666,E2 -1683.666} C_VEL
LIN {X 0,Y 580.305,Z 444.2,A -85,B 0,C 180,E1 -1685.684,E2 -1685.684} C_VEL
LIN {X 0,Y 580.273,Z 444.203,A -85,B 0,C 180,E1 -1687.947,E2 -1687.947} C_VEL
LIN {X 0,Y 580.302,Z 444.199,A -85,B 0,C 180,E1 -1690.914,E2 -1690.914} C_VEL
LIN {X 0,Y 580.273,Z 444.202,A -85,B 0,C 180,E1 -1693.825,E2 -1693.825} C_VEL
LIN {X 0,Y 580.331,Z 444.198,A -85,B 0,C 180,E1 -1695.983,E2 -1695.983} C_VEL
LIN {X 0,Y 580.311,Z 444.198,A -85,B 0,C 180,E1 -1698.827,E2 -1698.827} C_VEL
LIN {X 0,Y 580.333,Z 444.195,A -85,B 0,C 180,E1 -1701.644,E2 -1701.644} C_VEL
LIN {X 0,Y 580.323,Z 444.197,A -85,B 0,C 180,E1 -1704.44,E2 -1704.44} C_VEL
LIN {X 0,Y 580.341,Z 444.199,A -85,B 0,C 180,E1 -1707.224,E2 -1707.224} C_VEL
LIN {X 0,Y 580.358,Z 444.194,A -85,B 0,C 180,E1 -1710,E2 -1710} C_VEL
LIN {X 0,Y 580.339,Z 444.194,A -85,B 0,C 180,E1 -1712.777,E2 -1712.777} C_VEL
LIN {X 0,Y 580.326,Z 444.196,A -85,B 0,C 180,E1 -1715.56,E2 -1715.56} C_VEL
LIN {X 0,Y 580.329,Z 444.197,A -85,B 0,C 180,E1 -1717.655,E2 -1717.655} C_VEL
LIN {X 0,Y 580.305,Z 444.198,A -85,B 0,C 180,E1 -1720.467,E2 -1720.467} C_VEL
LIN {X 0,Y 580.309,Z 444.202,A -85,B 0,C 180,E1 -1722.591,E2 -1722.591} C_VEL
LIN {X 0,Y 580.291,Z 444.201,A -85,B 0,C 180,E1 -1724.734,E2 -1724.734} C_VEL
LIN {X 0,Y 580.295,Z 444.203,A -85,B 0,C 180,E1 -1727.625,E2 -1727.625} C_VEL
LIN {X 0,Y 580.293,Z 444.2,A -85,B 0,C 180,E1 -1729.823,E2 -1729.823} C_VEL
LIN {X 0,Y 580.276,Z 444.208,A -85,B 0,C 180,E1 -1732.053,E2 -1732.053} C_VEL
LIN {X 0,Y 580.312,Z 444.202,A -85,B 0,C 180,E1 -1735.08,E2 -1735.08} C_VEL
LIN {X 0,Y 580.302,Z 444.203,A -85,B 0,C 180,E1 -1738.186,E2 -1738.186} C_VEL
LIN {X 0,Y 580.289,Z 444.2,A -85,B 0,C 180,E1 -1740.694,E2 -1740.694} C_VEL
LIN {X 0,Y 580.307,Z 444.2,A -85,B 0,C 180,E1 -1743.316,E2 -1743.316} C_VEL
LIN {X 0,Y 580.252,Z 444.206,A -85,B 0,C 180,E1 -1745.756,E2 -1745.756} C_VEL
LIN {X 0,Y 580.291,Z 444.201,A -85,B 0,C 180,E1 -1748.146,E2 -1748.146} C_VEL
LIN {X 0,Y 580.302,Z 444.204,A -85,B 0,C 180,E1 -1750.843,E2 -1750.843} C_VEL
LIN {X 0,Y 580.278,Z 444.204,A -85,B 0,C 180,E1 -1753.658,E2 -1753.658} C_VEL
LIN {X 0,Y 580.283,Z 444.202,A -85,B 0,C 180,E1 -1756.609,E2 -1756.609} C_VEL
LIN {X 0,Y 580.302,Z 444.199,A -85,B 0,C 180,E1 -1759.156,E2 -1759.156} C_VEL
LIN {X 0,Y 580.292,Z 444.203,A -85,B 0,C 180,E1 -1761.927,E2 -1761.927} C_VEL
LIN {X 0,Y 580.23,Z 444.209,A -85,B 0,C 180,E1 -1764.451,E2 -1764.451} C_VEL
LIN {X 0,Y 580.193,Z 444.218,A -85,B 0,C 180,E1 -1765.457,E2 -1765.457} C_VEL
LIN {X 0,Y 580.144,Z 445.254,A -85,B 0,C 180,E1 -1766.708,E2 -1766.708} C_VEL
LIN {X 0,Y 580.132,Z 448.388,A -85,B 0,C 180,E1 -1769.415,E2 -1769.415} C_VEL
LIN {X 0,Y 580.135,Z 451.663,A -85,B 0,C 180,E1 -1772.172,E2 -1772.172} C_VEL
LIN {X 0,Y 580.088,Z 454.885,A -85,B 0,C 180,E1 -1774.91,E2 -1774.91} C_VEL
LIN {X 0,Y 580.076,Z 457.767,A -85,B 0,C 180,E1 -1777.188,E2 -1777.188} C_VEL
LIN {X 0,Y 580.087,Z 460.649,A -85,B 0,C 180,E1 -1779.43,E2 -1779.43} C_VEL
LIN {X 0,Y 580.042,Z 464.493,A -85,B 0,C 180,E1 -1782.367,E2 -1782.367} C_VEL
LIN {X 0,Y 580.057,Z 467.375,A -85,B 0,C 180,E1 -1784.541,E2 -1784.541} C_VEL
LIN {X 0,Y 580.073,Z 471.219,A -85,B 0,C 180,E1 -1787.403,E2 -1787.403} C_VEL
LIN {X 0,Y 580.075,Z 471.669,A -85,B 0,C 180,E1 -1787.737,E2 -1787.737} C_VEL
LIN {X 0,Y 580.774,Z 477.399,A -85,B 0,C 180,E1 -1787.885,E2 -1787.885} C_VEL
LIN {X 0,Y 580.698,Z 490.446,A -85,B 0,C 180,E1 -1788.26,E2 -1788.26} C_VEL
LIN {X 0,Y 580.598,Z 502.254,A -85,B 0,C 180,E1 -1788.735,E2 -1788.735} C_VEL
LIN {X 0,Y 580.516,Z 514.027,A -85,B 0,C 180,E1 -1789.361,E2 -1789.361} C_VEL
LIN {X 0,Y 580.39,Z 525.661,A -85,B 0,C 180,E1 -1790.151,E2 -1790.151} C_VEL
LIN {X 0,Y 580.308,Z 535.041,A -85,B 0,C 180,E1 -1790.941,E2 -1790.941} C_VEL
LIN {X 0,Y 580.251,Z 543.604,A -85,B 0,C 180,E1 -1791.818,E2 -1791.818} C_VEL
LIN {X 0,Y 580.205,Z 551.917,A -85,B 0,C 180,E1 -1792.868,E2 -1792.868} C_VEL
LIN {X 0,Y 580.14,Z 558.617,A -85,B 0,C 180,E1 -1793.915,E2 -1793.915} C_VEL
LIN {X 0,Y 580.053,Z 564.76,A -85,B 0,C 180,E1 -1795.135,E2 -1795.135} C_VEL
LIN {X 0,Y 580.11,Z 568.749,A -85,B 0,C 180,E1 -1796.179,E2 -1796.179} C_VEL
LIN {X 0,Y 580.043,Z 571.698,A -85,B 0,C 180,E1 -1797.222,E2 -1797.222} C_VEL
LIN {X 0,Y 580.038,Z 573.128,A -85,B 0,C 180,E1 -1797.917,E2 -1797.917} C_VEL
LIN {X 0,Y 580.041,Z 574.754,A -85,B 0,C 180,E1 -1799.306,E2 -1799.306} C_VEL
LIN {X 0,Y 580.038,Z 574.996,A -85,B 0,C 180,E1 -1800,E2 -1800} C_VEL
LIN {X 0,Y 580.04,Z 574.815,A -85,B 0,C 180,E1 -1800.694,E2 -1800.694} C_VEL
LIN {X 0,Y 580.037,Z 573.273,A -85,B 0,C 180,E1 -1802.083,E2 -1802.083} C_VEL
LIN {X 0,Y 580.044,Z 571.912,A -85,B 0,C 180,E1 -1802.778,E2 -1802.778} C_VEL
LIN {X 0,Y 580.11,Z 569.034,A -85,B 0,C 180,E1 -1803.82,E2 -1803.82} C_VEL
LIN {X 0,Y 580.053,Z 565.134,A -85,B 0,C 180,E1 -1804.865,E2 -1804.865} C_VEL
LIN {X 0,Y 580.162,Z 560.102,A -85,B 0,C 180,E1 -1805.91,E2 -1805.91} C_VEL
LIN {X 0,Y 580.158,Z 553.78,A -85,B 0,C 180,E1 -1806.958,E2 -1806.958} C_VEL
LIN {X 0,Y 580.241,Z 545.861,A -85,B 0,C 180,E1 -1808.007,E2 -1808.007} C_VEL
LIN {X 0,Y 580.308,Z 536.012,A -85,B 0,C 180,E1 -1809.058,E2 -1809.058} C_VEL
LIN {X 0,Y 580.408,Z 525.691,A -85,B 0,C 180,E1 -1809.936,E2 -1809.936} C_VEL
LIN {X 0,Y 580.502,Z 514.058,A -85,B 0,C 180,E1 -1810.728,E2 -1810.728} C_VEL
LIN {X 0,Y 580.602,Z 502.616,A -85,B 0,C 180,E1 -1811.338,E2 -1811.338} C_VEL
LIN {X 0,Y 580.678,Z 490.497,A -85,B 0,C 180,E1 -1811.829,E2 -1811.829} C_VEL
LIN {X 0,Y 580.779,Z 477.468,A -85,B 0,C 180,E1 -1812.204,E2 -1812.204} C_VEL
LIN {X 0,Y 580.09,Z 471.671,A -85,B 0,C 180,E1 -1812.352,E2 -1812.352} C_VEL
LIN {X 0,Y 580.047,Z 468.457,A -85,B 0,C 180,E1 -1814.74,E2 -1814.74} C_VEL
LIN {X 0,Y 580.066,Z 465.573,A -85,B 0,C 180,E1 -1816.905,E2 -1816.905} C_VEL
LIN {X 0,Y 580.064,Z 461.728,A -85,B 0,C 180,E1 -1819.831,E2 -1819.831} C_VEL
LIN {X 0,Y 580.046,Z 458.844,A -85,B 0,C 180,E1 -1822.062,E2 -1822.062} C_VEL
LIN {X 0,Y 580.097,Z 455.511,A -85,B 0,C 180,E1 -1824.681,E2 -1824.681} C_VEL
LIN {X 0,Y 580.089,Z 453.157,A -85,B 0,C 180,E1 -1826.633,E2 -1826.633} C_VEL
LIN {X 0,Y 580.154,Z 450.523,A -85,B 0,C 180,E1 -1829.283,E2 -1829.283} C_VEL
LIN {X 0,Y 580.214,Z 447.287,A -85,B 0,C 180,E1 -1832.206,E2 -1832.206} C_VEL
LIN {X 0,Y 580.201,Z 444.582,A -85,B 0,C 180,E1 -1834.702,E2 -1834.702} C_VEL
LIN {X 0,Y 580.268,Z 444.208,A -85,B 0,C 180,E1 -1836.404,E2 -1836.404} C_VEL
LIN {X 0,Y 580.302,Z 444.204,A -85,B 0,C 180,E1 -1839.186,E2 -1839.186} C_VEL
LIN {X 0,Y 580.318,Z 444.2,A -85,B 0,C 180,E1 -1841.766,E2 -1841.766} C_VEL
LIN {X 0,Y 580.273,Z 444.205,A -85,B 0,C 180,E1 -1844.626,E2 -1844.626} C_VEL
LIN {X 0,Y 580.289,Z 444.206,A -85,B 0,C 180,E1 -1847.628,E2 -1847.628} C_VEL
LIN {X 0,Y 580.299,Z 444.205,A -85,B 0,C 180,E1 -1850.067,E2 -1850.067} C_VEL
LIN {X 0,Y 580.324,Z 444.269,A -85,B 0,C 180,E1 -1853.173,E2 -1853.173} C_VEL
LIN {X 0,Y 580.752,Z 447.555,A -85,B 0,C 180,E1 -1854.488,E2 -1854.488} C_VEL
LIN {X 0,Y 580.634,Z 453.745,A -85,B 0,C 180,E1 -1856.635,E2 -1856.635} C_VEL
LIN {X 0,Y 580.576,Z 462.213,A -85,B 0,C 180,E1 -1859.257,E2 -1859.257} C_VEL
LIN {X 0,Y 580.528,Z 471.934,A -85,B 0,C 180,E1 -1862.099,E2 -1862.099} C_VEL
LIN {X 0,Y 580.45,Z 481.69,A -85,B 0,C 180,E1 -1864.927,E2 -1864.927} C_VEL
LIN {X 0,Y 580.369,Z 492.281,A -85,B 0,C 180,E1 -1867.951,E2 -1867.951} C_VEL
LIN {X 0,Y 580.268,Z 502.678,A -85,B 0,C 180,E1 -1870.858,E2 -1870.858} C_VEL
LIN {X 0,Y 580.222,Z 513.463,A -85,B 0,C 180,E1 -1873.824,E2 -1873.824} C_VEL
LIN {X 0,Y 580.186,Z 524.054,A -85,B 0,C 180,E1 -1876.694,E2 -1876.694} C_VEL
LIN {X 0,Y 580.146,Z 527.53,A -85,B 0,C 180,E1 -1877.627,E2 -1877.627} C_VEL
LIN {X 0,Y 580.814,Z 533.223,A -85,B 0,C 180,E1 -1877.753,E2 -1877.753} C_VEL
LIN {X 0,Y 580.737,Z 546.493,A -85,B 0,C 180,E1 -1878.083,E2 -1878.083} C_VEL
LIN {X 0,Y 580.659,Z 558.523,A -85,B 0,C 180,E1 -1878.525,E2 -1878.525} C_VEL
LIN {X 0,Y 580.531,Z 570.209,A -85,B 0,C 180,E1 -1879.096,E2 -1879.096} C_VEL
LIN {X 0,Y 580.447,Z 581.477,A -85,B 0,C 180,E1 -1879.8,E2 -1879.8} C_VEL
LIN {X 0,Y 580.352,Z 591.646,A -85,B 0,C 180,E1 -1880.591,E2 -1880.591} C_VEL
LIN {X 0,Y 580.279,Z 600.786,A -85,B 0,C 180,E1 -1881.468,E2 -1881.468} C_VEL
LIN {X 0,Y 580.199,Z 609.689,A -85,B 0,C 180,E1 -1882.518,E2 -1882.518} C_VEL
LIN {X 0,Y 580.12,Z 616.465,A -85,B 0,C 180,E1 -1883.505,E2 -1883.505} C_VEL
LIN {X 0,Y 580.139,Z 621.68,A -85,B 0,C 180,E1 -1884.438,E2 -1884.438} C_VEL
LIN {X 0,Y 580.108,Z 626.371,A -85,B 0,C 180,E1 -1885.483,E2 -1885.483} C_VEL
LIN {X 0,Y 580.123,Z 629.956,A -85,B 0,C 180,E1 -1886.527,E2 -1886.527} C_VEL
LIN {X 0,Y 580.043,Z 631.808,A -85,B 0,C 180,E1 -1887.222,E2 -1887.222} C_VEL
LIN {X 0,Y 580.038,Z 633.2,A -85,B 0,C 180,E1 -1887.917,E2 -1887.917} C_VEL
LIN {X 0,Y 580.04,Z 634.784,A -85,B 0,C 180,E1 -1889.306,E2 -1889.306} C_VEL
LIN {X 0,Y 580.037,Z 635,A -85,B 0,C 180,E1 -1890,E2 -1890} C_VEL
LIN {X 0,Y 580.047,Z 634.186,A -85,B 0,C 180,E1 -1891.388,E2 -1891.388} C_VEL
LIN {X 0,Y 580.038,Z 633.201,A -85,B 0,C 180,E1 -1892.083,E2 -1892.083} C_VEL
LIN {X 0,Y 580.043,Z 631.81,A -85,B 0,C 180,E1 -1892.778,E2 -1892.778} C_VEL
LIN {X 0,Y 580.109,Z 628.896,A -85,B 0,C 180,E1 -1893.821,E2 -1893.821} C_VEL
LIN {X 0,Y 580.054,Z 624.95,A -85,B 0,C 180,E1 -1894.865,E2 -1894.865} C_VEL
LIN {X 0,Y 580.139,Z 618.878,A -85,B 0,C 180,E1 -1896.085,E2 -1896.085} C_VEL
LIN {X 0,Y 580.184,Z 612.237,A -85,B 0,C 180,E1 -1897.132,E2 -1897.132} C_VEL
LIN {X 0,Y 580.25,Z 603.99,A -85,B 0,C 180,E1 -1898.182,E2 -1898.182} C_VEL
LIN {X 0,Y 580.308,Z 595.538,A -85,B 0,C 180,E1 -1899.058,E2 -1899.058} C_VEL
LIN {X 0,Y 580.417,Z 585.096,A -85,B 0,C 180,E1 -1899.936,E2 -1899.936} C_VEL
LIN {X 0,Y 580.506,Z 574.758,A -85,B 0,C 180,E1 -1900.639,E2 -1900.639} C_VEL
LIN {X 0,Y 580.584,Z 563.373,A -85,B 0,C 180,E1 -1901.258,E2 -1901.258} C_VEL
LIN {X 0,Y 580.675,Z 551.768,A -85,B 0,C 180,E1 -1901.741,E2 -1901.741} C_VEL
LIN {X 0,Y 580.776,Z 538.351,A -85,B 0,C 180,E1 -1902.137,E2 -1902.137} C_VEL
LIN {X 0,Y 580.612,Z 530.333,A -85,B 0,C 180,E1 -1902.307,E2 -1902.307} C_VEL
LIN {X 0,Y 580.146,Z 527.53,A -85,B 0,C 180,E1 -1902.373,E2 -1902.373} C_VEL
LIN {X 0,Y 580.226,Z 517.436,A -85,B 0,C 180,E1 -1905.095,E2 -1905.095} C_VEL
LIN {X 0,Y 580.253,Z 506.844,A -85,B 0,C 180,E1 -1907.99,E2 -1907.99} C_VEL
LIN {X 0,Y 580.344,Z 496.491,A -85,B 0,C 180,E1 -1910.864,E2 -1910.864} C_VEL
LIN {X 0,Y 580.404,Z 486.986,A -85,B 0,C 180,E1 -1913.553,E2 -1913.553} C_VEL
LIN {X 0,Y 580.455,Z 479.042,A -85,B 0,C 180,E1 -1915.841,E2 -1915.841} C_VEL
LIN {X 0,Y 580.509,Z 469.721,A -85,B 0,C 180,E1 -1918.569,E2 -1918.569} C_VEL
LIN {X 0,Y 580.607,Z 461.47,A -85,B 0,C 180,E1 -1921.017,E2 -1921.017} C_VEL
LIN {X 0,Y 580.731,Z 452.483,A -85,B 0,C 180,E1 -1923.827,E2 -1923.827} C_VEL
LIN {X 0,Y 580.662,Z 446.38,A -85,B 0,C 180,E1 -1925.813,E2 -1925.813} C_VEL
LIN {X 0,Y 580.311,Z 444.203,A -85,B 0,C 180,E1 -1926.591,E2 -1926.591} C_VEL
LIN {X 0,Y 580.31,Z 444.199,A -85,B 0,C 180,E1 -1929.187,E2 -1929.187} C_VEL
LIN {X 0,Y 580.283,Z 444.203,A -85,B 0,C 180,E1 -1931.769,E2 -1931.769} C_VEL
LIN {X 0,Y 580.269,Z 444.208,A -85,B 0,C 180,E1 -1934.626,E2 -1934.626} C_VEL
LIN {X 0,Y 580.285,Z 444.203,A -85,B 0,C 180,E1 -1937.294,E2 -1937.294} C_VEL
LIN {X 0,Y 580.285,Z 444.2,A -85,B 0,C 180,E1 -1940.066,E2 -1940.066} C_VEL
LIN {X 0,Y 580.301,Z 444.199,A -85,B 0,C 180,E1 -1943.066,E2 -1943.066} C_VEL
LIN {X 0,Y 580.319,Z 444.196,A -85,B 0,C 180,E1 -1946.145,E2 -1946.145} C_VEL
LIN {X 0,Y 580.279,Z 444.207,A -85,B 0,C 180,E1 -1948.615,E2 -1948.615} C_VEL
LIN {X 0,Y 580.295,Z 444.199,A -85,B 0,C 180,E1 -1951.024,E2 -1951.024} C_VEL
LIN {X 0,Y 580.294,Z 444.201,A -85,B 0,C 180,E1 -1953.666,E2 -1953.666} C_VEL
LIN {X 0,Y 580.302,Z 444.198,A -85,B 0,C 180,E1 -1955.684,E2 -1955.684} C_VEL
LIN {X 0,Y 580.278,Z 444.207,A -85,B 0,C 180,E1 -1957.948,E2 -1957.948} C_VEL
LIN {X 0,Y 580.322,Z 444.201,A -85,B 0,C 180,E1 -1960.914,E2 -1960.914} C_VEL
LIN {X 0,Y 580.282,Z 444.203,A -85,B 0,C 180,E1 -1963.826,E2 -1963.826} C_VEL
LIN {X 0,Y 580.329,Z 444.198,A -85,B 0,C 180,E1 -1965.983,E2 -1965.983} C_VEL
LIN {X 0,Y 580.308,Z 444.204,A -85,B 0,C 180,E1 -1968.827,E2 -1968.827} C_VEL
LIN {X 0,Y 580.331,Z 444.197,A -85,B 0,C 180,E1 -1971.644,E2 -1971.644} C_VEL
LIN {X 0,Y 580.325,Z 444.196,A -85,B 0,C 180,E1 -1974.44,E2 -1974.44} C_VEL
LIN {X 0,Y 580.343,Z 444.193,A -85,B 0,C 180,E1 -1977.224,E2 -1977.224} C_VEL
LIN {X 0,Y 580.356,Z 444.195,A -85,B 0,C 180,E1 -1980,E2 -1980} C_VEL
LIN {X 0,Y 580.347,Z 444.198,A -85,B 0,C 180,E1 -1982.777,E2 -1982.777} C_VEL
LIN {X 0,Y 580.324,Z 444.197,A -85,B 0,C 180,E1 -1985.56,E2 -1985.56} C_VEL
LIN {X 0,Y 580.336,Z 444.194,A -85,B 0,C 180,E1 -1988.356,E2 -1988.356} C_VEL
LIN {X 0,Y 580.303,Z 444.199,A -85,B 0,C 180,E1 -1991.191,E2 -1991.191} C_VEL
LIN {X 0,Y 580.33,Z 444.199,A -85,B 0,C 180,E1 -1994.017,E2 -1994.017} C_VEL
LIN {X 0,Y 580.316,Z 444.203,A -85,B 0,C 180,E1 -1996.914,E2 -1996.914} C_VEL
LIN {X 0,Y 580.308,Z 444.201,A -85,B 0,C 180,E1 -1999.822,E2 -1999.822} C_VEL
LIN {X 0,Y 580.287,Z 444.203,A -85,B 0,C 180,E1 -2001.333,E2 -2001.333} C_VEL
LIN {X 0,Y 579.59,Z 444.29,A -85,B 0,C 180,E1 -2001.912,E2 -2001.912} C_VEL
LIN {X 0,Y 576.713,Z 444.648,A -85,B 0,C 180,E1 -2002.852,E2 -2002.852} C_VEL
LIN {X 0,Y 574.318,Z 444.945,A -85,B 0,C 180,E1 -2003.608,E2 -2003.608} C_VEL
LIN {X 0,Y 573.319,Z 445.069,A -85,B 0,C 180,E1 -2004.192,E2 -2004.192} C_VEL
LIN {X 0,Y 573.253,Z 445.079,A -85,B 0,C 180,E1 -2004.389,E2 -2004.389} C_VEL
LIN {X 0,Y 573.253,Z 445.076,A -85,B 0,C 180,E1 -2006.976,E2 -2006.976} C_VEL
LIN {X 0,Y 573.25,Z 445.082,A -85,B 0,C 180,E1 -2009.488,E2 -2009.488} C_VEL
LIN {X 0,Y 573.259,Z 445.08,A -85,B 0,C 180,E1 -2012.645,E2 -2012.645} C_VEL
LIN {X 0,Y 573.257,Z 445.077,A -85,B 0,C 180,E1 -2015.185,E2 -2015.185} C_VEL
LIN {X 0,Y 573.239,Z 445.079,A -85,B 0,C 180,E1 -2017.808,E2 -2017.808} C_VEL
LIN {X 0,Y 573.248,Z 445.08,A -85,B 0,C 180,E1 -2020.525,E2 -2020.525} C_VEL
LIN {X 0,Y 573.251,Z 445.082,A -85,B 0,C 180,E1 -2023.358,E2 -2023.358} C_VEL
LIN {X 0,Y 573.247,Z 445.08,A -85,B 0,C 180,E1 -2026.331,E2 -2026.331} C_VEL
LIN {X 0,Y 573.232,Z 445.08,A -85,B 0,C 180,E1 -2028.543,E2 -2028.543} C_VEL
LIN {X 0,Y 573.246,Z 445.083,A -85,B 0,C 180,E1 -2031.299,E2 -2031.299} C_VEL
LIN {X 0,Y 573.242,Z 445.08,A -85,B 0,C 180,E1 -2034.015,E2 -2034.015} C_VEL
LIN {X 0,Y 573.274,Z 445.074,A -85,B 0,C 180,E1 -2036.518,E2 -2036.518} C_VEL
LIN {X 0,Y 573.232,Z 445.084,A -85,B 0,C 180,E1 -2039.118,E2 -2039.118} C_VEL
LIN {X 0,Y 573.239,Z 445.078,A -85,B 0,C 180,E1 -2041.436,E2 -2041.436} C_VEL
LIN {X 0,Y 573.258,Z 445.076,A -85,B 0,C 180,E1 -2044.59,E2 -2044.59} C_VEL
LIN {X 0,Y 573.239,Z 445.078,A -85,B 0,C 180,E1 -2047.662,E2 -2047.662} C_VEL
LIN {X 0,Y 573.271,Z 445.074,A -85,B 0,C 180,E1 -2050.67,E2 -2050.67} C_VEL
LIN {X 0,Y 573.247,Z 445.078,A -85,B 0,C 180,E1 -2053.622,E2 -2053.622} C_VEL
LIN {X 0,Y 573.279,Z 445.075,A -85,B 0,C 180,E1 -2055.807,E2 -2055.807} C_VEL
LIN {X 0,Y 573.269,Z 445.075,A -85,B 0,C 180,E1 -2058.745,E2 -2058.745} C_VEL
LIN {X 0,Y 573.289,Z 445.072,A -85,B 0,C 180,E1 -2061.541,E2 -2061.541} C_VEL
LIN {X 0,Y 573.29,Z 445.073,A -85,B 0,C 180,E1 -2064.372,E2 -2064.372} C_VEL
LIN {X 0,Y 573.317,Z 445.069,A -85,B 0,C 180,E1 -2067.893,E2 -2067.893} C_VEL
LIN {X 0,Y 573.333,Z 445.067,A -85,B 0,C 180,E1 -2070.702,E2 -2070.702} C_VEL
LIN {X 0,Y 573.306,Z 445.07,A -85,B 0,C 180,E1 -2072.811,E2 -2072.811} C_VEL
LIN {X 0,Y 573.294,Z 445.072,A -85,B 0,C 180,E1 -2075.628,E2 -2075.628} C_VEL
LIN {X 0,Y 573.277,Z 445.076,A -85,B 0,C 180,E1 -2077.75,E2 -2077.75} C_VEL
LIN {X 0,Y 573.272,Z 445.075,A -85,B 0,C 180,E1 -2080.597,E2 -2080.597} C_VEL
LIN {X 0,Y 573.269,Z 445.08,A -85,B 0,C 180,E1 -2082.749,E2 -2082.749} C_VEL
LIN {X 0,Y 573.238,Z 445.078,A -85,B 0,C 180,E1 -2084.92,E2 -2084.92} C_VEL
LIN {X 0,Y 573.247,Z 445.079,A -85,B 0,C 180,E1 -2087.849,E2 -2087.849} C_VEL
LIN {X 0,Y 573.248,Z 445.078,A -85,B 0,C 180,E1 -2090.077,E2 -2090.077} C_VEL
LIN {X 0,Y 573.241,Z 445.08,A -85,B 0,C 180,E1 -2092.338,E2 -2092.338} C_VEL
LIN {X 0,Y 573.26,Z 445.079,A -85,B 0,C 180,E1 -2095.41,E2 -2095.41} C_VEL
LIN {X 0,Y 573.253,Z 445.079,A -85,B 0,C 180,E1 -2098.028,E2 -2098.028} C_VEL
LIN {X 0,Y 573.252,Z 445.079,A -85,B 0,C 180,E1 -2100.176,E2 -2100.176} C_VEL
LIN {X 0,Y 573.258,Z 445.078,A -85,B 0,C 180,E1 -2102.645,E2 -2102.645} C_VEL
LIN {X 0,Y 573.214,Z 445.082,A -85,B 0,C 180,E1 -2105.188,E2 -2105.188} C_VEL
LIN {X 0,Y 573.239,Z 445.083,A -85,B 0,C 180,E1 -2107.808,E2 -2107.808} C_VEL
LIN {X 0,Y 573.249,Z 445.08,A -85,B 0,C 180,E1 -2110.525,E2 -2110.525} C_VEL
LIN {X 0,Y 573.242,Z 445.078,A -85,B 0,C 180,E1 -2113.359,E2 -2113.359} C_VEL
LIN {X 0,Y 573.25,Z 445.077,A -85,B 0,C 180,E1 -2116.331,E2 -2116.331} C_VEL
LIN {X 0,Y 573.249,Z 445.083,A -85,B 0,C 180,E1 -2118.544,E2 -2118.544} C_VEL
LIN {X 0,Y 573.243,Z 445.079,A -85,B 0,C 180,E1 -2121.298,E2 -2121.298} C_VEL
LIN {X 0,Y 573.197,Z 445.084,A -85,B 0,C 180,E1 -2123.947,E2 -2123.947} C_VEL
LIN {X 0,Y 573.119,Z 445.099,A -85,B 0,C 180,E1 -2125.661,E2 -2125.661} C_VEL
LIN {X 0,Y 573.077,Z 445.618,A -85,B 0,C 180,E1 -2126.505,E2 -2126.505} C_VEL
LIN {X 0,Y 573.06,Z 448.641,A -85,B 0,C 180,E1 -2129.147,E2 -2129.147} C_VEL
LIN {X 0,Y 573.066,Z 452.253,A -85,B 0,C 180,E1 -2132.223,E2 -2132.223} C_VEL
LIN {X 0,Y 573.018,Z 455.628,A -85,B 0,C 180,E1 -2135.177,E2 -2135.177} C_VEL
LIN {X 0,Y 572.956,Z 458.729,A -85,B 0,C 180,E1 -2137.65,E2 -2137.65} C_VEL
LIN {X 0,Y 572.987,Z 461.611,A -85,B 0,C 180,E1 -2139.913,E2 -2139.913} C_VEL
LIN {X 0,Y 572.991,Z 465.716,A -85,B 0,C 180,E1 -2143.08,E2 -2143.08} C_VEL
LIN {X 0,Y 572.988,Z 469.298,A -85,B 0,C 180,E1 -2145.8,E2 -2145.8} C_VEL
LIN {X 0,Y 573.01,Z 471.67,A -85,B 0,C 180,E1 -2147.583,E2 -2147.583} C_VEL
LIN {X 0,Y 573.827,Z 478.336,A -85,B 0,C 180,E1 -2147.758,E2 -2147.758} C_VEL
LIN {X 0,Y 573.741,Z 490.462,A -85,B 0,C 180,E1 -2148.115,E2 -2148.115} C_VEL
LIN {X 0,Y 573.642,Z 502.995,A -85,B 0,C 180,E1 -2148.631,E2 -2148.631} C_VEL
LIN {X 0,Y 573.542,Z 514.086,A -85,B 0,C 180,E1 -2149.233,E2 -2149.233} C_VEL
LIN {X 0,Y 573.394,Z 525.67,A -85,B 0,C 180,E1 -2150.03,E2 -2150.03} C_VEL
LIN {X 0,Y 573.287,Z 535.048,A -85,B 0,C 180,E1 -2150.83,E2 -2150.83} C_VEL
LIN {X 0,Y 573.202,Z 543.609,A -85,B 0,C 180,E1 -2151.717,E2 -2151.717} C_VEL
LIN {X 0,Y 573.138,Z 551.922,A -85,B 0,C 180,E1 -2152.779,E2 -2152.779} C_VEL
LIN {X 0,Y 573.065,Z 558.62,A -85,B 0,C 180,E1 -2153.84,E2 -2153.84} C_VEL
LIN {X 0,Y 572.963,Z 564.762,A -85,B 0,C 180,E1 -2155.074,E2 -2155.074} C_VEL
LIN {X 0,Y 573.015,Z 568.751,A -85,B 0,C 180,E1 -2156.132,E2 -2156.132} C_VEL
LIN {X 0,Y 572.959,Z 571.7,A -85,B 0,C 180,E1 -2157.188,E2 -2157.188} C_VEL
LIN {X 0,Y 572.938,Z 573.128,A -85,B 0,C 180,E1 -2157.891,E2 -2157.891} C_VEL
LIN {X 0,Y 572.942,Z 574.755,A -85,B 0,C 180,E1 -2159.297,E2 -2159.297} C_VEL
LIN {X 0,Y 572.938,Z 574.996,A -85,B 0,C 180,E1 -2160,E2 -2160} C_VEL
LIN {X 0,Y 572.94,Z 574.815,A -85,B 0,C 180,E1 -2160.703,E2 -2160.703} C_VEL
LIN {X 0,Y 572.937,Z 573.271,A -85,B 0,C 180,E1 -2162.109,E2 -2162.109} C_VEL
LIN {X 0,Y 572.96,Z 571.91,A -85,B 0,C 180,E1 -2162.812,E2 -2162.812} C_VEL
LIN {X 0,Y 573.015,Z 569.032,A -85,B 0,C 180,E1 -2163.868,E2 -2163.868} C_VEL
LIN {X 0,Y 572.963,Z 565.132,A -85,B 0,C 180,E1 -2164.926,E2 -2164.926} C_VEL
LIN {X 0,Y 573.076,Z 560.099,A -85,B 0,C 180,E1 -2165.983,E2 -2165.983} C_VEL
LIN {X 0,Y 573.083,Z 553.776,A -85,B 0,C 180,E1 -2167.044,E2 -2167.044} C_VEL
LIN {X 0,Y 573.175,Z 545.856,A -85,B 0,C 180,E1 -2168.106,E2 -2168.106} C_VEL
LIN {X 0,Y 573.287,Z 536.006,A -85,B 0,C 180,E1 -2169.17,E2 -2169.17} C_VEL
LIN {X 0,Y 573.41,Z 525.685,A -85,B 0,C 180,E1 -2170.059,E2 -2170.059} C_VEL
LIN {X 0,Y 573.505,Z 514.135,A -85,B 0,C 180,E1 -2170.855,E2 -2170.855} C_VEL
LIN {X 0,Y 573.638,Z 502.869,A -85,B 0,C 180,E1 -2171.466,E2 -2171.466} C_VEL
LIN {X 0,Y 573.724,Z 490.482,A -85,B 0,C 180,E1 -2171.975,E2 -2171.975} C_VEL
LIN {X 0,Y 573.844,Z 477.444,A -85,B 0,C 180,E1 -2172.354,E2 -2172.354} C_VEL
LIN {X 0,Y 572.981,Z 471.67,A -85,B 0,C 180,E1 -2172.507,E2 -2172.507} C_VEL
LIN {X 0,Y 572.961,Z 468.456,A -85,B 0,C 180,E1 -2174.927,E2 -2174.927} C_VEL
LIN {X 0,Y 572.976,Z 465.572,A -85,B 0,C 180,E1 -2177.12,E2 -2177.12} C_VEL
LIN {X 0,Y 572.987,Z 461.727,A -85,B 0,C 180,E1 -2180.086,E2 -2180.086} C_VEL
LIN {X 0,Y 572.99,Z 457.881,A -85,B 0,C 180,E1 -2183.11,E2 -2183.11} C_VEL
LIN {X 0,Y 573.005,Z 455.132,A -85,B 0,C 180,E1 -2185.422,E2 -2185.422} C_VEL
LIN {X 0,Y 573.082,Z 452.573,A -85,B 0,C 180,E1 -2187.996,E2 -2187.996} C_VEL
LIN {X 0,Y 573.118,Z 449.31,A -85,B 0,C 180,E1 -2191,E2 -2191} C_VEL
LIN {X 0,Y 573.173,Z 446.697,A -85,B 0,C 180,E1 -2193.51,E2 -2193.51} C_VEL
LIN {X 0,Y 573.166,Z 445.094,A -85,B 0,C 180,E1 -2195.191,E2 -2195.191} C_VEL
LIN {X 0,Y 573.24,Z 445.084,A -85,B 0,C 180,E1 -2197.807,E2 -2197.807} C_VEL
LIN {X 0,Y 573.247,Z 445.081,A -85,B 0,C 180,E1 -2200.525,E2 -2200.525} C_VEL
LIN {X 0,Y 573.251,Z 445.08,A -85,B 0,C 180,E1 -2203.358,E2 -2203.358} C_VEL
LIN {X 0,Y 573.247,Z 445.083,A -85,B 0,C 180,E1 -2206.331,E2 -2206.331} C_VEL
LIN {X 0,Y 573.278,Z 445.077,A -85,B 0,C 180,E1 -2209.477,E2 -2209.477} C_VEL
LIN {X 0,Y 573.239,Z 445.084,A -85,B 0,C 180,E1 -2212.192,E2 -2212.192} C_VEL
LIN {X 0,Y 573.279,Z 445.214,A -85,B 0,C 180,E1 -2212.894,E2 -2212.894} C_VEL
LIN {X 0,Y 573.817,Z 448.885,A -85,B 0,C 180,E1 -2214.425,E2 -2214.425} C_VEL
LIN {X 0,Y 573.663,Z 454.84,A -85,B 0,C 180,E1 -2216.544,E2 -2216.544} C_VEL
LIN {X 0,Y 573.575,Z 462.683,A -85,B 0,C 180,E1 -2219.061,E2 -2219.061} C_VEL
LIN {X 0,Y 573.486,Z 472.315,A -85,B 0,C 180,E1 -2221.928,E2 -2221.928} C_VEL
LIN {X 0,Y 573.423,Z 481.69,A -85,B 0,C 180,E1 -2224.598,E2 -2224.598} C_VEL
LIN {X 0,Y 573.364,Z 490.957,A -85,B 0,C 180,E1 -2227.287,E2 -2227.287} C_VEL
LIN {X 0,Y 573.262,Z 501.548,A -85,B 0,C 180,E1 -2230.297,E2 -2230.297} C_VEL
LIN {X 0,Y 573.175,Z 512.368,A -85,B 0,C 180,E1 -2233.316,E2 -2233.316} C_VEL
LIN {X 0,Y 573.123,Z 522.731,A -85,B 0,C 180,E1 -2236.165,E2 -2236.165} C_VEL
LIN {X 0,Y 573.107,Z 527.53,A -85,B 0,C 180,E1 -2237.473,E2 -2237.473} C_VEL
LIN {X 0,Y 573.88,Z 534.364,A -85,B 0,C 180,E1 -2237.625,E2 -2237.625} C_VEL
LIN {X 0,Y 573.787,Z 546.494,A -85,B 0,C 180,E1 -2237.937,E2 -2237.937} C_VEL
LIN {X 0,Y 573.693,Z 558.745,A -85,B 0,C 180,E1 -2238.393,E2 -2238.393} C_VEL
LIN {X 0,Y 573.556,Z 570.305,A -85,B 0,C 180,E1 -2238.967,E2 -2238.967} C_VEL
LIN {X 0,Y 573.424,Z 581.479,A -85,B 0,C 180,E1 -2239.674,E2 -2239.674} C_VEL
LIN {X 0,Y 573.308,Z 591.646,A -85,B 0,C 180,E1 -2240.474,E2 -2240.474} C_VEL
LIN {X 0,Y 573.215,Z 600.786,A -85,B 0,C 180,E1 -2241.362,E2 -2241.362} C_VEL
LIN {X 0,Y 573.142,Z 609.689,A -85,B 0,C 180,E1 -2242.425,E2 -2242.425} C_VEL
LIN {X 0,Y 573.051,Z 616.404,A -85,B 0,C 180,E1 -2243.415,E2 -2243.415} C_VEL
LIN {X 0,Y 573.07,Z 621.68,A -85,B 0,C 180,E1 -2244.37,E2 -2244.37} C_VEL
LIN {X 0,Y 573.029,Z 626.371,A -85,B 0,C 180,E1 -2245.427,E2 -2245.427} C_VEL
LIN {X 0,Y 573.022,Z 629.957,A -85,B 0,C 180,E1 -2246.484,E2 -2246.484} C_VEL
LIN {X 0,Y 572.959,Z 631.808,A -85,B 0,C 180,E1 -2247.188,E2 -2247.188} C_VEL
LIN {X 0,Y 572.938,Z 633.199,A -85,B 0,C 180,E1 -2247.891,E2 -2247.891} C_VEL
LIN {X 0,Y 572.941,Z 634.785,A -85,B 0,C 180,E1 -2249.297,E2 -2249.297} C_VEL
LIN {X 0,Y 572.938,Z 635,A -85,B 0,C 180,E1 -2250,E2 -2250} C_VEL
LIN {X 0,Y 572.946,Z 634.186,A -85,B 0,C 180,E1 -2251.406,E2 -2251.406} C_VEL
LIN {X 0,Y 572.938,Z 633.2,A -85,B 0,C 180,E1 -2252.109,E2 -2252.109} C_VEL
LIN {X 0,Y 572.959,Z 631.81,A -85,B 0,C 180,E1 -2252.812,E2 -2252.812} C_VEL
LIN {X 0,Y 573.014,Z 628.896,A -85,B 0,C 180,E1 -2253.868,E2 -2253.868} C_VEL
LIN {X 0,Y 572.963,Z 624.949,A -85,B 0,C 180,E1 -2254.926,E2 -2254.926} C_VEL
LIN {X 0,Y 573.064,Z 618.877,A -85,B 0,C 180,E1 -2256.16,E2 -2256.16} C_VEL
LIN {X 0,Y 573.119,Z 612.238,A -85,B 0,C 180,E1 -2257.221,E2 -2257.221} C_VEL
LIN {X 0,Y 573.201,Z 603.991,A -85,B 0,C 180,E1 -2258.283,E2 -2258.283} C_VEL
LIN {X 0,Y 573.287,Z 595.539,A -85,B 0,C 180,E1 -2259.17,E2 -2259.17} C_VEL
LIN {X 0,Y 573.42,Z 585.097,A -85,B 0,C 180,E1 -2260.058,E2 -2260.058} C_VEL
LIN {X 0,Y 573.548,Z 573.446,A -85,B 0,C 180,E1 -2260.852,E2 -2260.852} C_VEL
LIN {X 0,Y 573.653,Z 562.281,A -85,B 0,C 180,E1 -2261.447,E2 -2261.447} C_VEL
LIN {X 0,Y 573.738,Z 549.175,A -85,B 0,C 180,E1 -2261.974,E2 -2261.974} C_VEL
LIN {X 0,Y 573.842,Z 536.521,A -85,B 0,C 180,E1 -2262.331,E2 -2262.331} C_VEL
LIN {X 0,Y 573.722,Z 531.374,A -85,B 0,C 180,E1 -2262.438,E2 -2262.438} C_VEL
LIN {X 0,Y 573.106,Z 527.53,A -85,B 0,C 180,E1 -2262.527,E2 -2262.527} C_VEL
LIN {X 0,Y 573.162,Z 517.436,A -85,B 0,C 180,E1 -2265.285,E2 -2265.285} C_VEL
LIN {X 0,Y 573.215,Z 506.844,A -85,B 0,C 180,E1 -2268.219,E2 -2268.219} C_VEL
LIN {X 0,Y 573.309,Z 497.577,A -85,B 0,C 180,E1 -2270.824,E2 -2270.824} C_VEL
LIN {X 0,Y 573.371,Z 488.311,A -85,B 0,C 180,E1 -2273.476,E2 -2273.476} C_VEL
LIN {X 0,Y 573.461,Z 480.366,A -85,B 0,C 180,E1 -2275.79,E2 -2275.79} C_VEL
LIN {X 0,Y 573.501,Z 470.985,A -85,B 0,C 180,E1 -2278.55,E2 -2278.55} C_VEL
LIN {X 0,Y 573.635,Z 462.924,A -85,B 0,C 180,E1 -2280.969,E2 -2280.969} C_VEL
LIN {X 0,Y 573.794,Z 453.679,A -85,B 0,C 180,E1 -2283.903,E2 -2283.903} C_VEL
LIN {X 0,Y 573.759,Z 448.577,A -85,B 0,C 180,E1 -2285.579,E2 -2285.579} C_VEL
LIN {X 0,Y 573.265,Z 445.08,A -85,B 0,C 180,E1 -2286.812,E2 -2286.812} C_VEL
LIN {X 0,Y 573.25,Z 445.082,A -85,B 0,C 180,E1 -2289.607,E2 -2289.607} C_VEL
LIN {X 0,Y 573.242,Z 445.081,A -85,B 0,C 180,E1 -2292.641,E2 -2292.641} C_VEL
LIN {X 0,Y 573.242,Z 445.079,A -85,B 0,C 180,E1 -2295.667,E2 -2295.667} C_VEL
LIN {X 0,Y 573.247,Z 445.078,A -85,B 0,C 180,E1 -2298.544,E2 -2298.544} C_VEL
LIN {X 0,Y 573.241,Z 445.078,A -85,B 0,C 180,E1 -2301.298,E2 -2301.298} C_VEL
LIN {X 0,Y 573.217,Z 445.086,A -85,B 0,C 180,E1 -2304.018,E2 -2304.018} C_VEL
LIN {X 0,Y 573.271,Z 445.075,A -85,B 0,C 180,E1 -2306.518,E2 -2306.518} C_VEL
LIN {X 0,Y 573.231,Z 445.08,A -85,B 0,C 180,E1 -2309.118,E2 -2309.118} C_VEL
LIN {X 0,Y 573.24,Z 445.081,A -85,B 0,C 180,E1 -2311.436,E2 -2311.436} C_VEL
